LIN {X 0,Y 680.2,Z 809.06,A -85,B 0,C 180,E1 4290.744,E2 4290.744} C_VEL
LIN {X 0,Y 680.187,Z 809.06,A -85,B 0,C 180,E1 4295.606,E2 4295.606} C_VEL
LIN {X 0,Y 680.262,Z 809.06,A -85,B 0,C 180,E1 4300.538,E2 4300.538} C_VEL
LIN {X 0,Y 680.314,Z 809.425,A -85,B 0,C 180,E1 4305.507,E2 4305.507} C_VEL
LIN {X 0,Y 694.764,Z 845.315,A -85,B 0,C 180,E1 4307.71,E2 4307.71} C_VEL
LIN {X 0,Y 692.334,Z 893.553,A -85,B 0,C 180,E1 4309.75,E2 4309.75} C_VEL
LIN {X 0,Y 689.663,Z 937.812,A -85,B 0,C 180,E1 4312.208,E2 4312.208} C_VEL
LIN {X 0,Y 687.125,Z 980.915,A -85,B 0,C 180,E1 4315.269,E2 4315.269} C_VEL
LIN {X 0,Y 684.876,Z 1019.676,A -85,B 0,C 180,E1 4318.735,E2 4318.735} C_VEL
LIN {X 0,Y 683.218,Z 1052.318,A -85,B 0,C 180,E1 4322.376,E2 4322.376} C_VEL
LIN {X 0,Y 682.033,Z 1079.766,A -85,B 0,C 180,E1 4326.2,E2 4326.2} C_VEL
LIN {X 0,Y 681.334,Z 1102.128,A -85,B 0,C 180,E1 4330.219,E2 4330.219} C_VEL
LIN {X 0,Y 680.855,Z 1118.33,A -85,B 0,C 180,E1 4334.129,E2 4334.129} C_VEL
LIN {X 0,Y 680.765,Z 1129.59,A -85,B 0,C 180,E1 4338.103,E2 4338.103} C_VEL
LIN {X 0,Y 680.55,Z 1135.714,A -85,B 0,C 180,E1 4342.175,E2 4342.175} C_VEL
LIN {X 0,Y 680.543,Z 1137,A -85,B 0,C 180,E1 4344.951,E2 4344.951} C_VEL
LIN {X 0,Y 680.663,Z 1134.112,A -85,B 0,C 180,E1 4349.233,E2 4349.233} C_VEL
LIN {X 0,Y 680.799,Z 1126.558,A -85,B 0,C 180,E1 4353.076,E2 4353.076} C_VEL
LIN {X 0,Y 680.997,Z 1113.936,A -85,B 0,C 180,E1 4356.994,E2 4356.994} C_VEL
LIN {X 0,Y 681.399,Z 1096.802,A -85,B 0,C 180,E1 4360.757,E2 4360.757} C_VEL
LIN {X 0,Y 682.358,Z 1072.024,A -85,B 0,C 180,E1 4364.884,E2 4364.884} C_VEL
LIN {X 0,Y 683.721,Z 1042.519,A -85,B 0,C 180,E1 4368.71,E2 4368.71} C_VEL
LIN {X 0,Y 685.454,Z 1008.675,A -85,B 0,C 180,E1 4372.241,E2 4372.241} C_VEL
LIN {X 0,Y 687.791,Z 969.225,A -85,B 0,C 180,E1 4375.541,E2 4375.541} C_VEL
LIN {X 0,Y 690.35,Z 927.638,A -85,B 0,C 180,E1 4378.317,E2 4378.317} C_VEL
LIN {X 0,Y 692.87,Z 881.741,A -85,B 0,C 180,E1 4380.727,E2 4380.727} C_VEL
LIN {X 0,Y 694.585,Z 843.173,A -85,B 0,C 180,E1 4382.295,E2 4382.295} C_VEL
LIN {X 0,Y 680.289,Z 809.06,A -85,B 0,C 180,E1 4384.475,E2 4384.475} C_VEL
LIN {X 0,Y 680.236,Z 809.06,A -85,B 0,C 180,E1 4389.187,E2 4389.187} C_VEL
LIN {X 0,Y 680.252,Z 809.06,A -85,B 0,C 180,E1 4394.546,E2 4394.546} C_VEL
LIN {X 0,Y 680.62,Z 809.06,A -85,B 0,C 180,E1 4399.775,E2 4399.775} C_VEL
LIN {X 0,Y 680.649,Z 809.06,A -85,B 0,C 180,E1 4404.911,E2 4404.911} C_VEL
LIN {X 0,Y 680.652,Z 809.06,A -85,B 0,C 180,E1 4410.005,E2 4410.005} C_VEL
LIN {X 0,Y 680.742,Z 809.06,A -85,B 0,C 180,E1 4415.099,E2 4415.099} C_VEL
LIN {X 0,Y 680.549,Z 809.06,A -85,B 0,C 180,E1 4420.237,E2 4420.237} C_VEL
LIN {X 0,Y 680.532,Z 809.06,A -85,B 0,C 180,E1 4425.458,E2 4425.458} C_VEL
LIN {X 0,Y 680.453,Z 809.06,A -85,B 0,C 180,E1 4430.818,E2 4430.818} C_VEL
LIN {X 0,Y 680.319,Z 809.06,A -85,B 0,C 180,E1 4436.379,E2 4436.379} C_VEL
LIN {X 0,Y 680.313,Z 809.06,A -85,B 0,C 180,E1 4440.727,E2 4440.727} C_VEL
LIN {X 0,Y 680.298,Z 809.06,A -85,B 0,C 180,E1 4445.281,E2 4445.281} C_VEL
LIN {X 0,Y 680.16,Z 809.06,A -85,B 0,C 180,E1 4450.948,E2 4450.948} C_VEL
LIN {X 0,Y 680.352,Z 809.06,A -85,B 0,C 180,E1 4455.3,E2 4455.3} C_VEL
LIN {X 0,Y 680.213,Z 809.06,A -85,B 0,C 180,E1 4461.04,E2 4461.04} C_VEL
LIN {X 0,Y 680.177,Z 809.06,A -85,B 0,C 180,E1 4466.265,E2 4466.265} C_VEL
LIN {X 0,Y 680.337,Z 809.06,A -85,B 0,C 180,E1 4470.751,E2 4470.751} C_VEL
LIN {X 0,Y 680.434,Z 809.06,A -85,B 0,C 180,E1 4475.586,E2 4475.586} C_VEL
LIN {X 0,Y 680.513,Z 809.06,A -85,B 0,C 180,E1 4480.546,E2 4480.546} C_VEL
LIN {X 0,Y 680.474,Z 809.06,A -85,B 0,C 180,E1 4485.863,E2 4485.863} C_VEL
LIN {X 0,Y 680.596,Z 809.06,A -85,B 0,C 180,E1 4491.06,E2 4491.06} C_VEL
LIN {X 0,Y 680.727,Z 809.06,A -85,B 0,C 180,E1 4496.182,E2 4496.182} C_VEL
LIN {X 0,Y 680.902,Z 809.06,A -85,B 0,C 180,E1 4501.272,E2 4501.272} C_VEL
LIN {X 0,Y 680.599,Z 809.06,A -85,B 0,C 180,E1 4506.374,E2 4506.374} C_VEL
LIN {X 0,Y 680.537,Z 809.06,A -85,B 0,C 180,E1 4511.527,E2 4511.527} C_VEL
LIN {X 0,Y 680.557,Z 809.06,A -85,B 0,C 180,E1 4516.776,E2 4516.776} C_VEL
LIN {X 0,Y 680.391,Z 809.06,A -85,B 0,C 180,E1 4522.181,E2 4522.181} C_VEL
LIN {X 0,Y 680.331,Z 809.06,A -85,B 0,C 180,E1 4522.927,E2 4522.927} C_VEL
LIN {X 0,Y 676.369,Z 809.06,A -85,B 0,C 180,E1 4524.36,E2 4524.36} C_VEL
LIN {X 0,Y 672.401,Z 809.06,A -85,B 0,C 180,E1 4525.811,E2 4525.811} C_VEL
LIN {X 0,Y 672.352,Z 809.06,A -85,B 0,C 180,E1 4531.339,E2 4531.339} C_VEL
LIN {X 0,Y 672.336,Z 809.06,A -85,B 0,C 180,E1 4535.985,E2 4535.985} C_VEL
LIN {X 0,Y 672.291,Z 809.06,A -85,B 0,C 180,E1 4540.677,E2 4540.677} C_VEL
LIN {X 0,Y 672.415,Z 809.06,A -85,B 0,C 180,E1 4545.979,E2 4545.979} C_VEL
LIN {X 0,Y 672.345,Z 809.06,A -85,B 0,C 180,E1 4547.281,E2 4547.281} C_VEL
LIN {X 0,Y 674.931,Z 814.91,A -85,B 0,C 180,E1 4547.589,E2 4547.589} C_VEL
LIN {X 0,Y 692.454,Z 845.695,A -85,B 0,C 180,E1 4549.313,E2 4549.313} C_VEL
LIN {X 0,Y 691.569,Z 922.86,A -85,B 0,C 180,E1 4550.398,E2 4550.398} C_VEL
LIN {X 0,Y 689.719,Z 966.962,A -85,B 0,C 180,E1 4551.427,E2 4551.427} C_VEL
LIN {X 0,Y 687.547,Z 1012.993,A -85,B 0,C 180,E1 4553.033,E2 4553.033} C_VEL
LIN {X 0,Y 684.845,Z 1057.118,A -85,B 0,C 180,E1 4555.103,E2 4555.103} C_VEL
LIN {X 0,Y 682.1,Z 1099.687,A -85,B 0,C 180,E1 4557.663,E2 4557.663} C_VEL
LIN {X 0,Y 679.28,Z 1140.676,A -85,B 0,C 180,E1 4560.788,E2 4560.788} C_VEL
LIN {X 0,Y 677.093,Z 1175.037,A -85,B 0,C 180,E1 4564.02,E2 4564.02} C_VEL
LIN {X 0,Y 675.283,Z 1208.242,A -85,B 0,C 180,E1 4567.912,E2 4567.912} C_VEL
LIN {X 0,Y 674.008,Z 1233.927,A -85,B 0,C 180,E1 4571.702,E2 4571.702} C_VEL
LIN {X 0,Y 673.404,Z 1254.994,A -85,B 0,C 180,E1 4575.705,E2 4575.705} C_VEL
LIN {X 0,Y 673.092,Z 1270.402,A -85,B 0,C 180,E1 4579.649,E2 4579.649} C_VEL
LIN {X 0,Y 672.976,Z 1280.56,A -85,B 0,C 180,E1 4583.549,E2 4583.549} C_VEL
LIN {X 0,Y 672.892,Z 1285.871,A -85,B 0,C 180,E1 4587.421,E2 4587.421} C_VEL
LIN {X 0,Y 673.007,Z 1286.67,A -85,B 0,C 180,E1 4591.281,E2 4591.281} C_VEL
LIN {X 0,Y 672.834,Z 1282.919,A -85,B 0,C 180,E1 4595.149,E2 4595.149} C_VEL
LIN {X 0,Y 672.864,Z 1274.306,A -85,B 0,C 180,E1 4599.039,E2 4599.039} C_VEL
LIN {X 0,Y 673.22,Z 1262.369,A -85,B 0,C 180,E1 4602.563,E2 4602.563} C_VEL
LIN {X 0,Y 673.685,Z 1243.504,A -85,B 0,C 180,E1 4606.612,E2 4606.612} C_VEL
LIN {X 0,Y 674.721,Z 1219.785,A -85,B 0,C 180,E1 4610.494,E2 4610.494} C_VEL
LIN {X 0,Y 676.337,Z 1189.33,A -85,B 0,C 180,E1 4614.408,E2 4614.408} C_VEL
LIN {X 0,Y 678.339,Z 1155.606,A -85,B 0,C 180,E1 4617.885,E2 4617.885} C_VEL
LIN {X 0,Y 680.944,Z 1116.496,A -85,B 0,C 180,E1 4621.144,E2 4621.144} C_VEL
LIN {X 0,Y 683.675,Z 1073.955,A -85,B 0,C 180,E1 4623.959,E2 4623.959} C_VEL
LIN {X 0,Y 686.596,Z 1029.232,A -85,B 0,C 180,E1 4626.275,E2 4626.275} C_VEL
LIN {X 0,Y 689.056,Z 982.863,A -85,B 0,C 180,E1 4628.07,E2 4628.07} C_VEL
LIN {X 0,Y 691.01,Z 936.03,A -85,B 0,C 180,E1 4629.35,E2 4629.35} C_VEL
LIN {X 0,Y 692.232,Z 887.052,A -85,B 0,C 180,E1 4630.15,E2 4630.15} C_VEL
LIN {X 0,Y 691.991,Z 845.459,A -85,B 0,C 180,E1 4630.723,E2 4630.723} C_VEL
LIN {X 0,Y 672.601,Z 810.385,A -85,B 0,C 180,E1 4632.657,E2 4632.657} C_VEL
LIN {X 0,Y 672.495,Z 809.06,A -85,B 0,C 180,E1 4632.782,E2 4632.782} C_VEL
LIN {X 0,Y 672.304,Z 809.06,A -85,B 0,C 180,E1 4637.868,E2 4637.868} C_VEL
LIN {X 0,Y 672.275,Z 809.06,A -85,B 0,C 180,E1 4642.638,E2 4642.638} C_VEL
LIN {X 0,Y 672.238,Z 809.06,A -85,B 0,C 180,E1 4647.353,E2 4647.353} C_VEL
LIN {X 0,Y 672.328,Z 809.06,A -85,B 0,C 180,E1 4651.838,E2 4651.838} C_VEL
LIN {X 0,Y 672.2,Z 809.06,A -85,B 0,C 180,E1 4657.154,E2 4657.154} C_VEL
LIN {X 0,Y 672.233,Z 809.06,A -85,B 0,C 180,E1 4661.658,E2 4661.658} C_VEL
LIN {X 0,Y 672.415,Z 809.64,A -85,B 0,C 180,E1 4664.957,E2 4664.957} C_VEL
LIN {X 0,Y 688.239,Z 847.852,A -85,B 0,C 180,E1 4667.398,E2 4667.398} C_VEL
LIN {X 0,Y 685.564,Z 895.468,A -85,B 0,C 180,E1 4669.452,E2 4669.452} C_VEL
LIN {X 0,Y 682.602,Z 939.865,A -85,B 0,C 180,E1 4671.967,E2 4671.967} C_VEL
LIN {X 0,Y 679.837,Z 982.551,A -85,B 0,C 180,E1 4675.059,E2 4675.059} C_VEL
LIN {X 0,Y 677.362,Z 1021.021,A -85,B 0,C 180,E1 4678.562,E2 4678.562} C_VEL
LIN {X 0,Y 675.566,Z 1053.378,A -85,B 0,C 180,E1 4682.243,E2 4682.243} C_VEL
LIN {X 0,Y 674.272,Z 1080.621,A -85,B 0,C 180,E1 4686.11,E2 4686.11} C_VEL
LIN {X 0,Y 673.504,Z 1102.103,A -85,B 0,C 180,E1 4690.038,E2 4690.038} C_VEL
LIN {X 0,Y 673.032,Z 1118.204,A -85,B 0,C 180,E1 4693.965,E2 4693.965} C_VEL
LIN {X 0,Y 672.892,Z 1128.636,A -85,B 0,C 180,E1 4697.604,E2 4697.604} C_VEL
LIN {X 0,Y 672.719,Z 1134.648,A -85,B 0,C 180,E1 4701.061,E2 4701.061} C_VEL
LIN {X 0,Y 672.605,Z 1136.938,A -85,B 0,C 180,E1 4705.266,E2 4705.266} C_VEL
LIN {X 0,Y 672.791,Z 1133.635,A -85,B 0,C 180,E1 4709.609,E2 4709.609} C_VEL
LIN {X 0,Y 672.957,Z 1126.007,A -85,B 0,C 180,E1 4713.387,E2 4713.387} C_VEL
LIN {X 0,Y 673.212,Z 1113.275,A -85,B 0,C 180,E1 4717.3,E2 4717.3} C_VEL
LIN {X 0,Y 673.741,Z 1094.48,A -85,B 0,C 180,E1 4721.384,E2 4721.384} C_VEL
LIN {X 0,Y 674.716,Z 1070.906,A -85,B 0,C 180,E1 4725.291,E2 4725.291} C_VEL
LIN {X 0,Y 676.283,Z 1041.021,A -85,B 0,C 180,E1 4729.166,E2 4729.166} C_VEL
LIN {X 0,Y 678.193,Z 1007.742,A -85,B 0,C 180,E1 4732.647,E2 4732.647} C_VEL
LIN {X 0,Y 680.795,Z 968.271,A -85,B 0,C 180,E1 4735.965,E2 4735.965} C_VEL
LIN {X 0,Y 683.603,Z 926.623,A -85,B 0,C 180,E1 4738.754,E2 4738.754} C_VEL
LIN {X 0,Y 686.379,Z 880.658,A -85,B 0,C 180,E1 4741.173,E2 4741.173} C_VEL
LIN {X 0,Y 687.87,Z 845.761,A -85,B 0,C 180,E1 4742.623,E2 4742.623} C_VEL
LIN {X 0,Y 672.359,Z 809.06,A -85,B 0,C 180,E1 4745.019,E2 4745.019} C_VEL
LIN {X 0,Y 672.331,Z 809.06,A -85,B 0,C 180,E1 4750.716,E2 4750.716} C_VEL
LIN {X 0,Y 672.433,Z 809.06,A -85,B 0,C 180,E1 4755.694,E2 4755.694} C_VEL
LIN {X 0,Y 672.681,Z 809.06,A -85,B 0,C 180,E1 4760.959,E2 4760.959} C_VEL
LIN {X 0,Y 672.768,Z 809.06,A -85,B 0,C 180,E1 4766.142,E2 4766.142} C_VEL
LIN {X 0,Y 672.896,Z 809.06,A -85,B 0,C 180,E1 4771.292,E2 4771.292} C_VEL
LIN {X 0,Y 672.654,Z 809.06,A -85,B 0,C 180,E1 4776.454,E2 4776.454} C_VEL
LIN {X 0,Y 672.629,Z 809.06,A -85,B 0,C 180,E1 4781.67,E2 4781.67} C_VEL
LIN {X 0,Y 672.673,Z 809.06,A -85,B 0,C 180,E1 4786.985,E2 4786.985} C_VEL
LIN {X 0,Y 672.468,Z 809.06,A -85,B 0,C 180,E1 4792.463,E2 4792.463} C_VEL
LIN {X 0,Y 672.432,Z 809.06,A -85,B 0,C 180,E1 4796.713,E2 4796.713} C_VEL
LIN {X 0,Y 672.367,Z 809.06,A -85,B 0,C 180,E1 4801.356,E2 4801.356} C_VEL
LIN {X 0,Y 672.334,Z 809.06,A -85,B 0,C 180,E1 4805.997,E2 4805.997} C_VEL
LIN {X 0,Y 672.257,Z 809.06,A -85,B 0,C 180,E1 4810.687,E2 4810.687} C_VEL
LIN {X 0,Y 672.372,Z 809.06,A -85,B 0,C 180,E1 4815.842,E2 4815.842} C_VEL
LIN {X 0,Y 672.317,Z 809.06,A -85,B 0,C 180,E1 4821.003,E2 4821.003} C_VEL
LIN {X 0,Y 672.287,Z 809.06,A -85,B 0,C 180,E1 4826.275,E2 4826.275} C_VEL
LIN {X 0,Y 672.481,Z 809.06,A -85,B 0,C 180,E1 4831.846,E2 4831.846} C_VEL
LIN {X 0,Y 672.489,Z 809.06,A -85,B 0,C 180,E1 4837.122,E2 4837.122} C_VEL
LIN {X 0,Y 672.603,Z 809.06,A -85,B 0,C 180,E1 4841.669,E2 4841.669} C_VEL
LIN {X 0,Y 672.519,Z 809.06,A -85,B 0,C 180,E1 4847.017,E2 4847.017} C_VEL
LIN {X 0,Y 672.766,Z 809.06,A -85,B 0,C 180,E1 4852.256,E2 4852.256} C_VEL
LIN {X 0,Y 672.902,Z 809.06,A -85,B 0,C 180,E1 4857.426,E2 4857.426} C_VEL
LIN {X 0,Y 672.764,Z 809.06,A -85,B 0,C 180,E1 4862.575,E2 4862.575} C_VEL
LIN {X 0,Y 672.691,Z 809.06,A -85,B 0,C 180,E1 4866.449,E2 4866.449} C_VEL
LIN {X 0,Y 672.682,Z 809.06,A -85,B 0,C 180,E1 4870.353,E2 4870.353} C_VEL
LIN {X 0,Y 672.606,Z 809.06,A -85,B 0,C 180,E1 4875.64,E2 4875.64} C_VEL
LIN {X 0,Y 672.538,Z 809.06,A -85,B 0,C 180,E1 4881.068,E2 4881.068} C_VEL
LIN {X 0,Y 672.401,Z 809.06,A -85,B 0,C 180,E1 4885.811,E2 4885.811} C_VEL
LIN {X 0,Y 668.475,Z 809.06,A -85,B 0,C 180,E1 4887.268,E2 4887.268} C_VEL
LIN {X 0,Y 664.434,Z 809.06,A -85,B 0,C 180,E1 4888.742,E2 4888.742} C_VEL
LIN {X 0,Y 664.486,Z 809.06,A -85,B 0,C 180,E1 4893.076,E2 4893.076} C_VEL
LIN {X 0,Y 664.378,Z 809.06,A -85,B 0,C 180,E1 4897.884,E2 4897.884} C_VEL
LIN {X 0,Y 664.506,Z 809.06,A -85,B 0,C 180,E1 4903.302,E2 4903.302} C_VEL
LIN {X 0,Y 664.45,Z 809.06,A -85,B 0,C 180,E1 4906.65,E2 4906.65} C_VEL
LIN {X 0,Y 666.896,Z 814.808,A -85,B 0,C 180,E1 4906.953,E2 4906.953} C_VEL
LIN {X 0,Y 686.477,Z 848.997,A -85,B 0,C 180,E1 4908.928,E2 4908.928} C_VEL
LIN {X 0,Y 685.465,Z 922.835,A -85,B 0,C 180,E1 4909.974,E2 4909.974} C_VEL
LIN {X 0,Y 683.47,Z 967.502,A -85,B 0,C 180,E1 4911.026,E2 4911.026} C_VEL
LIN {X 0,Y 681.085,Z 1013.115,A -85,B 0,C 180,E1 4912.629,E2 4912.629} C_VEL
LIN {X 0,Y 678.207,Z 1056.587,A -85,B 0,C 180,E1 4914.68,E2 4914.68} C_VEL
LIN {X 0,Y 675.251,Z 1098.141,A -85,B 0,C 180,E1 4917.187,E2 4917.187} C_VEL
LIN {X 0,Y 672.226,Z 1138.223,A -85,B 0,C 180,E1 4920.234,E2 4920.234} C_VEL
LIN {X 0,Y 669.782,Z 1173.415,A -85,B 0,C 180,E1 4923.535,E2 4923.535} C_VEL
LIN {X 0,Y 667.651,Z 1206.126,A -85,B 0,C 180,E1 4927.366,E2 4927.366} C_VEL
LIN {X 0,Y 666.283,Z 1231.954,A -85,B 0,C 180,E1 4931.14,E2 4931.14} C_VEL
LIN {X 0,Y 665.611,Z 1251.057,A -85,B 0,C 180,E1 4934.679,E2 4934.679} C_VEL
LIN {X 0,Y 665.138,Z 1266.966,A -85,B 0,C 180,E1 4938.529,E2 4938.529} C_VEL
LIN {X 0,Y 664.972,Z 1277.702,A -85,B 0,C 180,E1 4942.158,E2 4942.158} C_VEL
LIN {X 0,Y 664.985,Z 1284.672,A -85,B 0,C 180,E1 4946.086,E2 4946.086} C_VEL
LIN {X 0,Y 664.95,Z 1287,A -85,B 0,C 180,E1 4949.995,E2 4949.995} C_VEL
LIN {X 0,Y 665.027,Z 1284.685,A -85,B 0,C 180,E1 4953.903,E2 4953.903} C_VEL
LIN {X 0,Y 664.965,Z 1277.728,A -85,B 0,C 180,E1 4957.831,E2 4957.831} C_VEL
LIN {X 0,Y 665.261,Z 1265.849,A -85,B 0,C 180,E1 4961.79,E2 4961.79} C_VEL
LIN {X 0,Y 665.675,Z 1248.748,A -85,B 0,C 180,E1 4965.801,E2 4965.801} C_VEL
LIN {X 0,Y 666.57,Z 1227.725,A -85,B 0,C 180,E1 4969.528,E2 4969.528} C_VEL
LIN {X 0,Y 668.057,Z 1199.843,A -85,B 0,C 180,E1 4973.444,E2 4973.444} C_VEL
LIN {X 0,Y 670.119,Z 1168.064,A -85,B 0,C 180,E1 4977.004,E2 4977.004} C_VEL
LIN {X 0,Y 672.789,Z 1131.27,A -85,B 0,C 180,E1 4980.354,E2 4980.354} C_VEL
LIN {X 0,Y 675.867,Z 1089.063,A -85,B 0,C 180,E1 4983.409,E2 4983.409} C_VEL
LIN {X 0,Y 678.951,Z 1046.719,A -85,B 0,C 180,E1 4985.837,E2 4985.837} C_VEL
LIN {X 0,Y 681.717,Z 1002.725,A -85,B 0,C 180,E1 4987.775,E2 4987.775} C_VEL
LIN {X 0,Y 684.002,Z 957.416,A -85,B 0,C 180,E1 4989.252,E2 4989.252} C_VEL
LIN {X 0,Y 685.728,Z 911.796,A -85,B 0,C 180,E1 4990.23,E2 4990.23} C_VEL
LIN {X 0,Y 686.126,Z 848.928,A -85,B 0,C 180,E1 4991.099,E2 4991.099} C_VEL
LIN {X 0,Y 664.669,Z 810.286,A -85,B 0,C 180,E1 4993.292,E2 4993.292} C_VEL
LIN {X 0,Y 664.559,Z 809.06,A -85,B 0,C 180,E1 4993.448,E2 4993.448} C_VEL
LIN {X 0,Y 664.342,Z 809.06,A -85,B 0,C 180,E1 4998.731,E2 4998.731} C_VEL
LIN {X 0,Y 664.376,Z 809.06,A -85,B 0,C 180,E1 5003.749,E2 5003.749} C_VEL
LIN {X 0,Y 664.333,Z 809.06,A -85,B 0,C 180,E1 5008.458,E2 5008.458} C_VEL
LIN {X 0,Y 664.421,Z 809.06,A -85,B 0,C 180,E1 5012.946,E2 5012.946} C_VEL
LIN {X 0,Y 664.412,Z 809.06,A -85,B 0,C 180,E1 5018.804,E2 5018.804} C_VEL
LIN {X 0,Y 664.425,Z 809.363,A -85,B 0,C 180,E1 5024.368,E2 5024.368} C_VEL
LIN {X 0,Y 681.715,Z 851.229,A -85,B 0,C 180,E1 5027.114,E2 5027.114} C_VEL
LIN {X 0,Y 678.769,Z 897.923,A -85,B 0,C 180,E1 5029.174,E2 5029.174} C_VEL
LIN {X 0,Y 675.505,Z 943.111,A -85,B 0,C 180,E1 5031.801,E2 5031.801} C_VEL
LIN {X 0,Y 672.55,Z 984.171,A -85,B 0,C 180,E1 5034.844,E2 5034.844} C_VEL
LIN {X 0,Y 669.858,Z 1022.355,A -85,B 0,C 180,E1 5038.384,E2 5038.384} C_VEL
LIN {X 0,Y 667.884,Z 1054.448,A -85,B 0,C 180,E1 5042.106,E2 5042.106} C_VEL
LIN {X 0,Y 666.543,Z 1080.442,A -85,B 0,C 180,E1 5045.854,E2 5045.854} C_VEL
LIN {X 0,Y 665.705,Z 1101.84,A -85,B 0,C 180,E1 5049.801,E2 5049.801} C_VEL
LIN {X 0,Y 665.167,Z 1118.084,A -85,B 0,C 180,E1 5053.799,E2 5053.799} C_VEL
LIN {X 0,Y 664.972,Z 1129.577,A -85,B 0,C 180,E1 5057.934,E2 5057.934} C_VEL
LIN {X 0,Y 664.799,Z 1135.004,A -85,B 0,C 180,E1 5061.324,E2 5061.324} C_VEL
LIN {X 0,Y 664.704,Z 1136.864,A -85,B 0,C 180,E1 5065.588,E2 5065.588} C_VEL
LIN {X 0,Y 664.776,Z 1135.08,A -85,B 0,C 180,E1 5068.51,E2 5068.51} C_VEL
LIN {X 0,Y 665.011,Z 1128.8,A -85,B 0,C 180,E1 5072.323,E2 5072.323} C_VEL
LIN {X 0,Y 665.166,Z 1117.778,A -85,B 0,C 180,E1 5076.2,E2 5076.2} C_VEL
LIN {X 0,Y 665.561,Z 1103.198,A -85,B 0,C 180,E1 5079.816,E2 5079.816} C_VEL
LIN {X 0,Y 666.338,Z 1082.447,A -85,B 0,C 180,E1 5083.726,E2 5083.726} C_VEL
LIN {X 0,Y 667.692,Z 1056.685,A -85,B 0,C 180,E1 5087.519,E2 5087.519} C_VEL
LIN {X 0,Y 669.71,Z 1024.273,A -85,B 0,C 180,E1 5091.327,E2 5091.327} C_VEL
LIN {X 0,Y 672.295,Z 987.168,A -85,B 0,C 180,E1 5094.817,E2 5094.817} C_VEL
LIN {X 0,Y 675.29,Z 947.344,A -85,B 0,C 180,E1 5097.821,E2 5097.821} C_VEL
LIN {X 0,Y 678.42,Z 904.103,A -85,B 0,C 180,E1 5100.411,E2 5100.411} C_VEL
LIN {X 0,Y 681.233,Z 861.151,A -85,B 0,C 180,E1 5102.405,E2 5102.405} C_VEL
LIN {X 0,Y 681.663,Z 849.788,A -85,B 0,C 180,E1 5102.861,E2 5102.861} C_VEL
LIN {X 0,Y 664.402,Z 809.06,A -85,B 0,C 180,E1 5105.602,E2 5105.602} C_VEL
LIN {X 0,Y 664.404,Z 809.06,A -85,B 0,C 180,E1 5110.059,E2 5110.059} C_VEL
LIN {X 0,Y 664.518,Z 809.06,A -85,B 0,C 180,E1 5115.52,E2 5115.52} C_VEL
LIN {X 0,Y 664.771,Z 809.06,A -85,B 0,C 180,E1 5120.85,E2 5120.85} C_VEL
LIN {X 0,Y 664.88,Z 809.06,A -85,B 0,C 180,E1 5126.096,E2 5126.096} C_VEL
LIN {X 0,Y 665.002,Z 809.06,A -85,B 0,C 180,E1 5131.307,E2 5131.307} C_VEL
LIN {X 0,Y 664.755,Z 809.06,A -85,B 0,C 180,E1 5136.531,E2 5136.531} C_VEL
LIN {X 0,Y 664.716,Z 809.06,A -85,B 0,C 180,E1 5141.811,E2 5141.811} C_VEL
LIN {X 0,Y 664.725,Z 809.06,A -85,B 0,C 180,E1 5147.313,E2 5147.313} C_VEL
LIN {X 0,Y 664.556,Z 809.06,A -85,B 0,C 180,E1 5152.745,E2 5152.745} C_VEL
LIN {X 0,Y 664.504,Z 809.06,A -85,B 0,C 180,E1 5157.527,E2 5157.527} C_VEL
LIN {X 0,Y 664.521,Z 809.06,A -85,B 0,C 180,E1 5163.081,E2 5163.081} C_VEL
LIN {X 0,Y 664.36,Z 809.06,A -85,B 0,C 180,E1 5167.893,E2 5167.893} C_VEL
LIN {X 0,Y 664.475,Z 809.06,A -85,B 0,C 180,E1 5173.31,E2 5173.31} C_VEL
LIN {X 0,Y 664.317,Z 809.06,A -85,B 0,C 180,E1 5178.731,E2 5178.731} C_VEL
LIN {X 0,Y 664.359,Z 809.06,A -85,B 0,C 180,E1 5183.749,E2 5183.749} C_VEL
LIN {X 0,Y 664.381,Z 809.06,A -85,B 0,C 180,E1 5188.461,E2 5188.461} C_VEL
LIN {X 0,Y 664.609,Z 809.06,A -85,B 0,C 180,E1 5192.955,E2 5192.955} C_VEL
LIN {X 0,Y 664.634,Z 809.06,A -85,B 0,C 180,E1 5198.67,E2 5198.67} C_VEL
LIN {X 0,Y 664.686,Z 809.06,A -85,B 0,C 180,E1 5204.17,E2 5204.17} C_VEL
LIN {X 0,Y 664.804,Z 809.06,A -85,B 0,C 180,E1 5209.524,E2 5209.524} C_VEL
LIN {X 0,Y 664.815,Z 809.06,A -85,B 0,C 180,E1 5214.784,E2 5214.784} C_VEL
LIN {X 0,Y 664.929,Z 809.06,A -85,B 0,C 180,E1 5219.708,E2 5219.708} C_VEL
LIN {X 0,Y 664.955,Z 809.06,A -85,B 0,C 180,E1 5223.909,E2 5223.909} C_VEL
LIN {X 0,Y 664.854,Z 809.06,A -85,B 0,C 180,E1 5229.154,E2 5229.154} C_VEL
LIN {X 0,Y 664.687,Z 809.06,A -85,B 0,C 180,E1 5234.481,E2 5234.481} C_VEL
LIN {X 0,Y 664.679,Z 809.06,A -85,B 0,C 180,E1 5238.558,E2 5238.558} C_VEL
LIN {X 0,Y 664.548,Z 809.06,A -85,B 0,C 180,E1 5242.739,E2 5242.739} C_VEL
LIN {X 0,Y 664.443,Z 809.06,A -85,B 0,C 180,E1 5247.5,E2 5247.5} C_VEL
LIN {X 0,Y 664.434,Z 809.06,A -85,B 0,C 180,E1 5248.742,E2 5248.742} C_VEL
LIN {X 0,Y 660.457,Z 809.06,A -85,B 0,C 180,E1 5250.217,E2 5250.217} C_VEL
LIN {X 0,Y 656.542,Z 809.06,A -85,B 0,C 180,E1 5251.709,E2 5251.709} C_VEL
LIN {X 0,Y 656.493,Z 809.06,A -85,B 0,C 180,E1 5256.757,E2 5256.757} C_VEL
LIN {X 0,Y 656.531,Z 809.06,A -85,B 0,C 180,E1 5262.558,E2 5262.558} C_VEL
LIN {X 0,Y 656.603,Z 809.06,A -85,B 0,C 180,E1 5266.019,E2 5266.019} C_VEL
LIN {X 0,Y 659.009,Z 814.762,A -85,B 0,C 180,E1 5266.309,E2 5266.309} C_VEL
LIN {X 0,Y 680.523,Z 852.366,A -85,B 0,C 180,E1 5268.536,E2 5268.536} C_VEL
LIN {X 0,Y 679.352,Z 923.994,A -85,B 0,C 180,E1 5269.565,E2 5269.565} C_VEL
LIN {X 0,Y 677.255,Z 967.989,A -85,B 0,C 180,E1 5270.615,E2 5270.615} C_VEL
LIN {X 0,Y 674.723,Z 1012.719,A -85,B 0,C 180,E1 5272.196,E2 5272.196} C_VEL
LIN {X 0,Y 671.609,Z 1056.2,A -85,B 0,C 180,E1 5274.258,E2 5274.258} C_VEL
LIN {X 0,Y 668.269,Z 1098.966,A -85,B 0,C 180,E1 5276.858,E2 5276.858} C_VEL
LIN {X 0,Y 664.943,Z 1139.603,A -85,B 0,C 180,E1 5279.998,E2 5279.998} C_VEL
LIN {X 0,Y 662.248,Z 1175.04,A -85,B 0,C 180,E1 5283.393,E2 5283.393} C_VEL
LIN {X 0,Y 659.946,Z 1207.625,A -85,B 0,C 180,E1 5287.289,E2 5287.289} C_VEL
LIN {X 0,Y 658.545,Z 1232.261,A -85,B 0,C 180,E1 5290.963,E2 5290.963} C_VEL
LIN {X 0,Y 657.726,Z 1252.321,A -85,B 0,C 180,E1 5294.768,E2 5294.768} C_VEL
LIN {X 0,Y 657.282,Z 1268.123,A -85,B 0,C 180,E1 5298.726,E2 5298.726} C_VEL
LIN {X 0,Y 657.129,Z 1279.211,A -85,B 0,C 180,E1 5302.729,E2 5302.729} C_VEL
LIN {X 0,Y 657.08,Z 1284.672,A -85,B 0,C 180,E1 5306.039,E2 5306.039} C_VEL
LIN {X 0,Y 657.075,Z 1287,A -85,B 0,C 180,E1 5309.995,E2 5309.995} C_VEL
LIN {X 0,Y 657.119,Z 1284.685,A -85,B 0,C 180,E1 5313.95,E2 5313.95} C_VEL
LIN {X 0,Y 657.07,Z 1277.725,A -85,B 0,C 180,E1 5317.926,E2 5317.926} C_VEL
LIN {X 0,Y 657.398,Z 1265.85,A -85,B 0,C 180,E1 5321.933,E2 5321.933} C_VEL
LIN {X 0,Y 657.839,Z 1249.826,A -85,B 0,C 180,E1 5325.778,E2 5325.778} C_VEL
LIN {X 0,Y 658.799,Z 1228.696,A -85,B 0,C 180,E1 5329.611,E2 5329.611} C_VEL
LIN {X 0,Y 660.348,Z 1201.517,A -85,B 0,C 180,E1 5333.512,E2 5333.512} C_VEL
LIN {X 0,Y 662.594,Z 1170.029,A -85,B 0,C 180,E1 5337.13,E2 5337.13} C_VEL
LIN {X 0,Y 665.676,Z 1131.248,A -85,B 0,C 180,E1 5340.715,E2 5340.715} C_VEL
LIN {X 0,Y 668.977,Z 1089.446,A -85,B 0,C 180,E1 5343.773,E2 5343.773} C_VEL
LIN {X 0,Y 672.36,Z 1046.704,A -85,B 0,C 180,E1 5346.245,E2 5346.245} C_VEL
LIN {X 0,Y 675.412,Z 1001.915,A -85,B 0,C 180,E1 5348.224,E2 5348.224} C_VEL
LIN {X 0,Y 677.847,Z 957.042,A -85,B 0,C 180,E1 5349.689,E2 5349.689} C_VEL
LIN {X 0,Y 679.724,Z 910.77,A -85,B 0,C 180,E1 5350.678,E2 5350.678} C_VEL
LIN {X 0,Y 680.189,Z 852.119,A -85,B 0,C 180,E1 5351.492,E2 5351.492} C_VEL
LIN {X 0,Y 656.877,Z 810.783,A -85,B 0,C 180,E1 5353.928,E2 5353.928} C_VEL
LIN {X 0,Y 656.682,Z 809.06,A -85,B 0,C 180,E1 5354.019,E2 5354.019} C_VEL
LIN {X 0,Y 656.404,Z 809.06,A -85,B 0,C 180,E1 5359.868,E2 5359.868} C_VEL
LIN {X 0,Y 656.433,Z 809.06,A -85,B 0,C 180,E1 5364.868,E2 5364.868} C_VEL
LIN {X 0,Y 656.424,Z 809.06,A -85,B 0,C 180,E1 5369.575,E2 5369.575} C_VEL
LIN {X 0,Y 656.491,Z 809.06,A -85,B 0,C 180,E1 5374.067,E2 5374.067} C_VEL
LIN {X 0,Y 656.516,Z 809.06,A -85,B 0,C 180,E1 5379.804,E2 5379.804} C_VEL
LIN {X 0,Y 656.454,Z 809.14,A -85,B 0,C 180,E1 5383.762,E2 5383.762} C_VEL
LIN {X 0,Y 675.009,Z 852.682,A -85,B 0,C 180,E1 5386.731,E2 5386.731} C_VEL
LIN {X 0,Y 671.989,Z 900.519,A -85,B 0,C 180,E1 5388.899,E2 5388.899} C_VEL
LIN {X 0,Y 668.407,Z 946.346,A -85,B 0,C 180,E1 5391.632,E2 5391.632} C_VEL
LIN {X 0,Y 665.282,Z 985.787,A -85,B 0,C 180,E1 5394.624,E2 5394.624} C_VEL
LIN {X 0,Y 662.477,Z 1022.118,A -85,B 0,C 180,E1 5398.039,E2 5398.039} C_VEL
LIN {X 0,Y 660.299,Z 1054.255,A -85,B 0,C 180,E1 5401.803,E2 5401.803} C_VEL
LIN {X 0,Y 658.776,Z 1081.294,A -85,B 0,C 180,E1 5405.759,E2 5405.759} C_VEL
LIN {X 0,Y 657.816,Z 1103.23,A -85,B 0,C 180,E1 5409.92,E2 5409.92} C_VEL
LIN {X 0,Y 657.269,Z 1119.137,A -85,B 0,C 180,E1 5413.968,E2 5413.968} C_VEL
LIN {X 0,Y 657.083,Z 1130.05,A -85,B 0,C 180,E1 5418.085,E2 5418.085} C_VEL
LIN {X 0,Y 656.848,Z 1135.326,A -85,B 0,C 180,E1 5421.595,E2 5421.595} C_VEL
LIN {X 0,Y 656.768,Z 1136.782,A -85,B 0,C 180,E1 5425.92,E2 5425.92} C_VEL
LIN {X 0,Y 657.077,Z 1132.658,A -85,B 0,C 180,E1 5430.391,E2 5430.391} C_VEL
LIN {X 0,Y 657.333,Z 1123.249,A -85,B 0,C 180,E1 5434.586,E2 5434.586} C_VEL
LIN {X 0,Y 657.69,Z 1107.865,A -85,B 0,C 180,E1 5438.948,E2 5438.948} C_VEL
LIN {X 0,Y 658.354,Z 1087.417,A -85,B 0,C 180,E1 5443.095,E2 5443.095} C_VEL
LIN {X 0,Y 659.813,Z 1061.64,A -85,B 0,C 180,E1 5447.122,E2 5447.122} C_VEL
LIN {X 0,Y 661.772,Z 1030.892,A -85,B 0,C 180,E1 5450.923,E2 5450.923} C_VEL
LIN {X 0,Y 664.441,Z 996.32,A -85,B 0,C 180,E1 5454.374,E2 5454.374} C_VEL
LIN {X 0,Y 667.578,Z 957.329,A -85,B 0,C 180,E1 5457.504,E2 5457.504} C_VEL
LIN {X 0,Y 670.863,Z 916.52,A -85,B 0,C 180,E1 5460.128,E2 5460.128} C_VEL
LIN {X 0,Y 673.925,Z 873.439,A -85,B 0,C 180,E1 5462.302,E2 5462.302} C_VEL
LIN {X 0,Y 674.788,Z 852.086,A -85,B 0,C 180,E1 5463.22,E2 5463.22} C_VEL
LIN {X 0,Y 658.078,Z 813.864,A -85,B 0,C 180,E1 5465.864,E2 5465.864} C_VEL
LIN {X 0,Y 656.419,Z 809.06,A -85,B 0,C 180,E1 5466.25,E2 5466.25} C_VEL
LIN {X 0,Y 656.429,Z 809.06,A -85,B 0,C 180,E1 5471.206,E2 5471.206} C_VEL
LIN {X 0,Y 656.655,Z 809.06,A -85,B 0,C 180,E1 5476.702,E2 5476.702} C_VEL
LIN {X 0,Y 656.916,Z 809.06,A -85,B 0,C 180,E1 5482.073,E2 5482.073} C_VEL
LIN {X 0,Y 657.028,Z 809.06,A -85,B 0,C 180,E1 5487.369,E2 5487.369} C_VEL
LIN {X 0,Y 656.898,Z 809.06,A -85,B 0,C 180,E1 5492.642,E2 5492.642} C_VEL
LIN {X 0,Y 656.849,Z 809.06,A -85,B 0,C 180,E1 5496.61,E2 5496.61} C_VEL
LIN {X 0,Y 656.827,Z 809.06,A -85,B 0,C 180,E1 5501.955,E2 5501.955} C_VEL
LIN {X 0,Y 656.827,Z 809.06,A -85,B 0,C 180,E1 5507.407,E2 5507.407} C_VEL
LIN {X 0,Y 656.644,Z 809.06,A -85,B 0,C 180,E1 5513.035,E2 5513.035} C_VEL
LIN {X 0,Y 656.597,Z 809.06,A -85,B 0,C 180,E1 5517.41,E2 5517.41} C_VEL
LIN {X 0,Y 656.553,Z 809.06,A -85,B 0,C 180,E1 5521.967,E2 5521.967} C_VEL
LIN {X 0,Y 656.48,Z 809.06,A -85,B 0,C 180,E1 5526.766,E2 5526.766} C_VEL
LIN {X 0,Y 656.498,Z 809.06,A -85,B 0,C 180,E1 5532.566,E2 5532.566} C_VEL
LIN {X 0,Y 656.393,Z 809.06,A -85,B 0,C 180,E1 5537.455,E2 5537.455} C_VEL
LIN {X 0,Y 656.423,Z 809.06,A -85,B 0,C 180,E1 5541.575,E2 5541.575} C_VEL
LIN {X 0,Y 656.394,Z 809.06,A -85,B 0,C 180,E1 5546.464,E2 5546.464} C_VEL
LIN {X 0,Y 656.569,Z 809.06,A -85,B 0,C 180,E1 5551.101,E2 5551.101} C_VEL
LIN {X 0,Y 656.695,Z 809.06,A -85,B 0,C 180,E1 5555.534,E2 5555.534} C_VEL
LIN {X 0,Y 656.759,Z 809.06,A -85,B 0,C 180,E1 5561.211,E2 5561.211} C_VEL
LIN {X 0,Y 656.744,Z 809.06,A -85,B 0,C 180,E1 5565.341,E2 5565.341} C_VEL
LIN {X 0,Y 656.887,Z 809.06,A -85,B 0,C 180,E1 5570.735,E2 5570.735} C_VEL
LIN {X 0,Y 657.022,Z 809.06,A -85,B 0,C 180,E1 5576.044,E2 5576.044} C_VEL
LIN {X 0,Y 657.232,Z 809.06,A -85,B 0,C 180,E1 5581.318,E2 5581.318} C_VEL
LIN {X 0,Y 656.887,Z 809.06,A -85,B 0,C 180,E1 5586.605,E2 5586.605} C_VEL
LIN {X 0,Y 656.843,Z 809.06,A -85,B 0,C 180,E1 5590.605,E2 5590.605} C_VEL
LIN {X 0,Y 656.789,Z 809.06,A -85,B 0,C 180,E1 5596.026,E2 5596.026} C_VEL
LIN {X 0,Y 656.675,Z 809.06,A -85,B 0,C 180,E1 5601.602,E2 5601.602} C_VEL
LIN {X 0,Y 656.554,Z 809.06,A -85,B 0,C 180,E1 5606.147,E2 5606.147} C_VEL
LIN {X 0,Y 656.542,Z 809.06,A -85,B 0,C 180,E1 5611.709,E2 5611.709} C_VEL
LIN {X 0,Y 652.541,Z 809.06,A -85,B 0,C 180,E1 5613.199,E2 5613.199} C_VEL
LIN {X 0,Y 648.553,Z 809.06,A -85,B 0,C 180,E1 5614.708,E2 5614.708} C_VEL
LIN {X 0,Y 648.484,Z 809.06,A -85,B 0,C 180,E1 5619.733,E2 5619.733} C_VEL
LIN {X 0,Y 648.645,Z 809.06,A -85,B 0,C 180,E1 5625.166,E2 5625.166} C_VEL
LIN {X 0,Y 648.659,Z 809.06,A -85,B 0,C 180,E1 5625.334,E2 5625.334} C_VEL
LIN {X 0,Y 651.222,Z 814.867,A -85,B 0,C 180,E1 5625.652,E2 5625.652} C_VEL
LIN {X 0,Y 674.551,Z 856.408,A -85,B 0,C 180,E1 5628.143,E2 5628.143} C_VEL
LIN {X 0,Y 673.288,Z 925.327,A -85,B 0,C 180,E1 5629.153,E2 5629.153} C_VEL
LIN {X 0,Y 671.037,Z 969.026,A -85,B 0,C 180,E1 5630.211,E2 5630.211} C_VEL
LIN {X 0,Y 668.285,Z 1013.712,A -85,B 0,C 180,E1 5631.815,E2 5631.815} C_VEL
LIN {X 0,Y 664.881,Z 1057.759,A -85,B 0,C 180,E1 5633.932,E2 5633.932} C_VEL
LIN {X 0,Y 661.279,Z 1100.163,A -85,B 0,C 180,E1 5636.55,E2 5636.55} C_VEL
LIN {X 0,Y 657.617,Z 1141.697,A -85,B 0,C 180,E1 5639.82,E2 5639.82} C_VEL
LIN {X 0,Y 654.674,Z 1176.943,A -85,B 0,C 180,E1 5643.279,E2 5643.279} C_VEL
LIN {X 0,Y 652.254,Z 1209.683,A -85,B 0,C 180,E1 5647.286,E2 5647.286} C_VEL
LIN {X 0,Y 650.636,Z 1235.774,A -85,B 0,C 180,E1 5651.348,E2 5651.348} C_VEL
LIN {X 0,Y 649.851,Z 1256.521,A -85,B 0,C 180,E1 5655.519,E2 5655.519} C_VEL
LIN {X 0,Y 649.415,Z 1270.403,A -85,B 0,C 180,E1 5659.267,E2 5659.267} C_VEL
LIN {X 0,Y 649.257,Z 1280.56,A -85,B 0,C 180,E1 5663.312,E2 5663.312} C_VEL
LIN {X 0,Y 649.202,Z 1285.871,A -85,B 0,C 180,E1 5667.326,E2 5667.326} C_VEL
LIN {X 0,Y 649.334,Z 1286.67,A -85,B 0,C 180,E1 5671.328,E2 5671.328} C_VEL
LIN {X 0,Y 649.193,Z 1282.919,A -85,B 0,C 180,E1 5675.337,E2 5675.337} C_VEL
LIN {X 0,Y 649.236,Z 1274.305,A -85,B 0,C 180,E1 5679.371,E2 5679.371} C_VEL
LIN {X 0,Y 649.706,Z 1260.73,A -85,B 0,C 180,E1 5683.443,E2 5683.443} C_VEL
LIN {X 0,Y 650.665,Z 1240.504,A -85,B 0,C 180,E1 5687.802,E2 5687.802} C_VEL
LIN {X 0,Y 652.1,Z 1214.292,A -85,B 0,C 180,E1 5692.051,E2 5692.051} C_VEL
LIN {X 0,Y 654.122,Z 1184.531,A -85,B 0,C 180,E1 5695.872,E2 5695.872} C_VEL
LIN {X 0,Y 657.114,Z 1147.943,A -85,B 0,C 180,E1 5699.623,E2 5699.623} C_VEL
LIN {X 0,Y 660.477,Z 1108.698,A -85,B 0,C 180,E1 5702.834,E2 5702.834} C_VEL
LIN {X 0,Y 664.199,Z 1065.637,A -85,B 0,C 180,E1 5705.639,E2 5705.639} C_VEL
LIN {X 0,Y 667.713,Z 1019.573,A -85,B 0,C 180,E1 5707.941,E2 5707.941} C_VEL
LIN {X 0,Y 670.774,Z 972.341,A -85,B 0,C 180,E1 5709.696,E2 5709.696} C_VEL
LIN {X 0,Y 673.123,Z 923.651,A -85,B 0,C 180,E1 5710.895,E2 5710.895} C_VEL
LIN {X 0,Y 674.287,Z 855.34,A -85,B 0,C 180,E1 5711.892,E2 5711.892} C_VEL
LIN {X 0,Y 650.355,Z 813.837,A -85,B 0,C 180,E1 5714.438,E2 5714.438} C_VEL
LIN {X 0,Y 648.675,Z 809.06,A -85,B 0,C 180,E1 5714.712,E2 5714.712} C_VEL
LIN {X 0,Y 648.489,Z 809.06,A -85,B 0,C 180,E1 5720.25,E2 5720.25} C_VEL
LIN {X 0,Y 648.537,Z 809.06,A -85,B 0,C 180,E1 5724.625,E2 5724.625} C_VEL
LIN {X 0,Y 648.536,Z 809.06,A -85,B 0,C 180,E1 5729.539,E2 5729.539} C_VEL
LIN {X 0,Y 648.58,Z 809.06,A -85,B 0,C 180,E1 5733.727,E2 5733.727} C_VEL
LIN {X 0,Y 648.573,Z 809.06,A -85,B 0,C 180,E1 5739.545,E2 5739.545} C_VEL
LIN {X 0,Y 648.532,Z 809.327,A -85,B 0,C 180,E1 5743.152,E2 5743.152} C_VEL
LIN {X 0,Y 667.981,Z 854.525,A -85,B 0,C 180,E1 5746.334,E2 5746.334} C_VEL
LIN {X 0,Y 668.313,Z 862.82,A -85,B 0,C 180,E1 5746.73,E2 5746.73} C_VEL
LIN {X 0,Y 664.695,Z 908.875,A -85,B 0,C 180,E1 5748.942,E2 5748.942} C_VEL
LIN {X 0,Y 661.031,Z 951.864,A -85,B 0,C 180,E1 5751.621,E2 5751.621} C_VEL
LIN {X 0,Y 657.532,Z 993.077,A -85,B 0,C 180,E1 5754.891,E2 5754.891} C_VEL
LIN {X 0,Y 654.495,Z 1029.46,A -85,B 0,C 180,E1 5758.511,E2 5758.511} C_VEL
LIN {X 0,Y 652.288,Z 1060.244,A -85,B 0,C 180,E1 5762.323,E2 5762.323} C_VEL
LIN {X 0,Y 650.624,Z 1085.945,A -85,B 0,C 180,E1 5766.333,E2 5766.333} C_VEL
LIN {X 0,Y 649.854,Z 1106.123,A -85,B 0,C 180,E1 5770.381,E2 5770.381} C_VEL
LIN {X 0,Y 649.321,Z 1121.194,A -85,B 0,C 180,E1 5774.486,E2 5774.486} C_VEL
LIN {X 0,Y 649.182,Z 1130.653,A -85,B 0,C 180,E1 5778.313,E2 5778.313} C_VEL
LIN {X 0,Y 648.933,Z 1135.597,A -85,B 0,C 180,E1 5781.872,E2 5781.872} C_VEL
LIN {X 0,Y 648.908,Z 1136.701,A -85,B 0,C 180,E1 5786.258,E2 5786.258} C_VEL
LIN {X 0,Y 649.204,Z 1132.089,A -85,B 0,C 180,E1 5790.799,E2 5790.799} C_VEL
LIN {X 0,Y 649.419,Z 1122.25,A -85,B 0,C 180,E1 5795.055,E2 5795.055} C_VEL
LIN {X 0,Y 649.835,Z 1107.57,A -85,B 0,C 180,E1 5799.195,E2 5799.195} C_VEL
LIN {X 0,Y 650.622,Z 1087.102,A -85,B 0,C 180,E1 5803.375,E2 5803.375} C_VEL
LIN {X 0,Y 652.198,Z 1060.828,A -85,B 0,C 180,E1 5807.511,E2 5807.511} C_VEL
LIN {X 0,Y 654.425,Z 1030.239,A -85,B 0,C 180,E1 5811.311,E2 5811.311} C_VEL
LIN {X 0,Y 657.268,Z 995.515,A -85,B 0,C 180,E1 5814.802,E2 5814.802} C_VEL
LIN {X 0,Y 660.726,Z 956.363,A -85,B 0,C 180,E1 5817.959,E2 5817.959} C_VEL
LIN {X 0,Y 664.295,Z 914.859,A -85,B 0,C 180,E1 5820.632,E2 5820.632} C_VEL
LIN {X 0,Y 667.676,Z 871.291,A -85,B 0,C 180,E1 5822.818,E2 5822.818} C_VEL
LIN {X 0,Y 668.464,Z 855.709,A -85,B 0,C 180,E1 5823.49,E2 5823.49} C_VEL
LIN {X 0,Y 652.399,Z 818.527,A -85,B 0,C 180,E1 5826.14,E2 5826.14} C_VEL
LIN {X 0,Y 648.508,Z 809.06,A -85,B 0,C 180,E1 5826.804,E2 5826.804} C_VEL
LIN {X 0,Y 648.531,Z 809.06,A -85,B 0,C 180,E1 5830.968,E2 5830.968} C_VEL
LIN {X 0,Y 648.727,Z 809.06,A -85,B 0,C 180,E1 5836.536,E2 5836.536} C_VEL
LIN {X 0,Y 649.024,Z 809.06,A -85,B 0,C 180,E1 5841.976,E2 5841.976} C_VEL
LIN {X 0,Y 649.151,Z 809.06,A -85,B 0,C 180,E1 5847.337,E2 5847.337} C_VEL
LIN {X 0,Y 649.002,Z 809.06,A -85,B 0,C 180,E1 5852.674,E2 5852.674} C_VEL
LIN {X 0,Y 648.96,Z 809.06,A -85,B 0,C 180,E1 5856.691,E2 5856.691} C_VEL
LIN {X 0,Y 648.937,Z 809.06,A -85,B 0,C 180,E1 5862.102,E2 5862.102} C_VEL
LIN {X 0,Y 648.922,Z 809.06,A -85,B 0,C 180,E1 5867.626,E2 5867.626} C_VEL
LIN {X 0,Y 648.707,Z 809.06,A -85,B 0,C 180,E1 5873.333,E2 5873.333} C_VEL
LIN {X 0,Y 648.66,Z 809.06,A -85,B 0,C 180,E1 5877.774,E2 5877.774} C_VEL
LIN {X 0,Y 648.609,Z 809.06,A -85,B 0,C 180,E1 5883.003,E2 5883.003} C_VEL
LIN {X 0,Y 648.493,Z 809.06,A -85,B 0,C 180,E1 5887.609,E2 5887.609} C_VEL
LIN {X 0,Y 648.591,Z 809.06,A -85,B 0,C 180,E1 5892.51,E2 5892.51} C_VEL
LIN {X 0,Y 648.49,Z 809.06,A -85,B 0,C 180,E1 5897.492,E2 5897.492} C_VEL
LIN {X 0,Y 648.471,Z 809.06,A -85,B 0,C 180,E1 5902.713,E2 5902.713} C_VEL
LIN {X 0,Y 648.496,Z 809.06,A -85,B 0,C 180,E1 5907.596,E2 5907.596} C_VEL
LIN {X 0,Y 648.75,Z 809.06,A -85,B 0,C 180,E1 5912.273,E2 5912.273} C_VEL
LIN {X 0,Y 648.762,Z 809.06,A -85,B 0,C 180,E1 5916.676,E2 5916.676} C_VEL
LIN {X 0,Y 648.868,Z 809.06,A -85,B 0,C 180,E1 5922.379,E2 5922.379} C_VEL
LIN {X 0,Y 648.892,Z 809.06,A -85,B 0,C 180,E1 5927.995,E2 5927.995} C_VEL
LIN {X 0,Y 649.066,Z 809.06,A -85,B 0,C 180,E1 5933.316,E2 5933.316} C_VEL
LIN {X 0,Y 649.08,Z 809.06,A -85,B 0,C 180,E1 5938.667,E2 5938.667} C_VEL
LIN {X 0,Y 649.091,Z 809.06,A -85,B 0,C 180,E1 5942.669,E2 5942.669} C_VEL
LIN {X 0,Y 649,Z 809.06,A -85,B 0,C 180,E1 5946.685,E2 5946.685} C_VEL
LIN {X 0,Y 648.9,Z 809.06,A -85,B 0,C 180,E1 5952.098,E2 5952.098} C_VEL
LIN {X 0,Y 648.876,Z 809.06,A -85,B 0,C 180,E1 5957.622,E2 5957.622} C_VEL
LIN {X 0,Y 648.697,Z 809.06,A -85,B 0,C 180,E1 5963.327,E2 5963.327} C_VEL
LIN {X 0,Y 648.597,Z 809.06,A -85,B 0,C 180,E1 5967.771,E2 5967.771} C_VEL
LIN {X 0,Y 648.588,Z 809.06,A -85,B 0,C 180,E1 5972.986,E2 5972.986} C_VEL
LIN {X 0,Y 648.553,Z 809.06,A -85,B 0,C 180,E1 5974.708,E2 5974.708} C_VEL
LIN {X 0,Y 647.276,Z 809.06,A -85,B 0,C 180,E1 5975.474,E2 5975.474} C_VEL
LIN {X 0,Y 640.656,Z 809.06,A -85,B 0,C 180,E1 5977.555,E2 5977.555} C_VEL
LIN {X 0,Y 640.582,Z 809.06,A -85,B 0,C 180,E1 5977.752,E2 5977.752} C_VEL
LIN {X 0,Y 640.715,Z 809.06,A -85,B 0,C 180,E1 5983.15,E2 5983.15} C_VEL
LIN {X 0,Y 640.759,Z 809.06,A -85,B 0,C 180,E1 5984.672,E2 5984.672} C_VEL
LIN {X 0,Y 643.264,Z 814.825,A -85,B 0,C 180,E1 5984.966,E2 5984.966} C_VEL
LIN {X 0,Y 668.445,Z 858.177,A -85,B 0,C 180,E1 5987.697,E2 5987.697} C_VEL
LIN {X 0,Y 667.215,Z 927.86,A -85,B 0,C 180,E1 5988.757,E2 5988.757} C_VEL
LIN {X 0,Y 664.738,Z 971.795,A -85,B 0,C 180,E1 5989.852,E2 5989.852} C_VEL
LIN {X 0,Y 661.613,Z 1017.452,A -85,B 0,C 180,E1 5991.543,E2 5991.543} C_VEL
LIN {X 0,Y 657.879,Z 1062.346,A -85,B 0,C 180,E1 5993.765,E2 5993.765} C_VEL
LIN {X 0,Y 654.079,Z 1103.672,A -85,B 0,C 180,E1 5996.41,E2 5996.41} C_VEL
LIN {X 0,Y 650.197,Z 1144.832,A -85,B 0,C 180,E1 5999.728,E2 5999.728} C_VEL
LIN {X 0,Y 646.967,Z 1180.428,A -85,B 0,C 180,E1 6003.34,E2 6003.34} C_VEL
LIN {X 0,Y 644.552,Z 1211.348,A -85,B 0,C 180,E1 6007.238,E2 6007.238} C_VEL
LIN {X 0,Y 642.798,Z 1237.866,A -85,B 0,C 180,E1 6011.492,E2 6011.492} C_VEL
LIN {X 0,Y 642.002,Z 1257.984,A -85,B 0,C 180,E1 6015.686,E2 6015.686} C_VEL
LIN {X 0,Y 641.507,Z 1272.344,A -85,B 0,C 180,E1 6019.819,E2 6019.819} C_VEL
LIN {X 0,Y 641.402,Z 1281.776,A -85,B 0,C 180,E1 6023.909,E2 6023.909} C_VEL
LIN {X 0,Y 641.298,Z 1285.871,A -85,B 0,C 180,E1 6027.293,E2 6027.293} C_VEL
LIN {X 0,Y 641.432,Z 1286.669,A -85,B 0,C 180,E1 6031.344,E2 6031.344} C_VEL
LIN {X 0,Y 641.296,Z 1282.919,A -85,B 0,C 180,E1 6035.403,E2 6035.403} C_VEL
LIN {X 0,Y 641.39,Z 1274.304,A -85,B 0,C 180,E1 6039.487,E2 6039.487} C_VEL
LIN {X 0,Y 641.865,Z 1260.731,A -85,B 0,C 180,E1 6043.61,E2 6043.61} C_VEL
LIN {X 0,Y 642.887,Z 1240.502,A -85,B 0,C 180,E1 6048.025,E2 6048.025} C_VEL
LIN {X 0,Y 644.453,Z 1214.294,A -85,B 0,C 180,E1 6052.326,E2 6052.326} C_VEL
LIN {X 0,Y 646.666,Z 1184.529,A -85,B 0,C 180,E1 6056.193,E2 6056.193} C_VEL
LIN {X 0,Y 649.898,Z 1147.936,A -85,B 0,C 180,E1 6059.986,E2 6059.986} C_VEL
LIN {X 0,Y 653.512,Z 1109.024,A -85,B 0,C 180,E1 6063.203,E2 6063.203} C_VEL
LIN {X 0,Y 657.539,Z 1065.921,A -85,B 0,C 180,E1 6066.038,E2 6066.038} C_VEL
LIN {X 0,Y 661.379,Z 1019.19,A -85,B 0,C 180,E1 6068.388,E2 6068.388} C_VEL
LIN {X 0,Y 664.647,Z 972.341,A -85,B 0,C 180,E1 6070.136,E2 6070.136} C_VEL
LIN {X 0,Y 667.204,Z 922.813,A -85,B 0,C 180,E1 6071.355,E2 6071.355} C_VEL
LIN {X 0,Y 668.098,Z 858.151,A -85,B 0,C 180,E1 6072.33,E2 6072.33} C_VEL
LIN {X 0,Y 643.046,Z 814.612,A -85,B 0,C 180,E1 6075.053,E2 6075.053} C_VEL
LIN {X 0,Y 640.73,Z 809.06,A -85,B 0,C 180,E1 6075.286,E2 6075.286} C_VEL
LIN {X 0,Y 640.564,Z 809.06,A -85,B 0,C 180,E1 6081.11,E2 6081.11} C_VEL
LIN {X 0,Y 640.587,Z 809.06,A -85,B 0,C 180,E1 6085.639,E2 6085.639} C_VEL
LIN {X 0,Y 640.625,Z 809.06,A -85,B 0,C 180,E1 6090.765,E2 6090.765} C_VEL
LIN {X 0,Y 640.614,Z 809.06,A -85,B 0,C 180,E1 6094.877,E2 6094.877} C_VEL
LIN {X 0,Y 640.631,Z 809.06,A -85,B 0,C 180,E1 6100.718,E2 6100.718} C_VEL
LIN {X 0,Y 640.628,Z 809.482,A -85,B 0,C 180,E1 6102.522,E2 6102.522} C_VEL
LIN {X 0,Y 660.074,Z 853.997,A -85,B 0,C 180,E1 6105.76,E2 6105.76} C_VEL
LIN {X 0,Y 662.15,Z 860.931,A -85,B 0,C 180,E1 6106.22,E2 6106.22} C_VEL
LIN {X 0,Y 658.273,Z 906.888,A -85,B 0,C 180,E1 6108.413,E2 6108.413} C_VEL
LIN {X 0,Y 654.332,Z 950.291,A -85,B 0,C 180,E1 6111.116,E2 6111.116} C_VEL
LIN {X 0,Y 650.558,Z 990.914,A -85,B 0,C 180,E1 6114.335,E2 6114.335} C_VEL
LIN {X 0,Y 647.249,Z 1027.751,A -85,B 0,C 180,E1 6117.993,E2 6117.993} C_VEL
LIN {X 0,Y 644.713,Z 1060.049,A -85,B 0,C 180,E1 6122.014,E2 6122.014} C_VEL
LIN {X 0,Y 642.928,Z 1085.774,A -85,B 0,C 180,E1 6126.07,E2 6126.07} C_VEL
LIN {X 0,Y 642.034,Z 1105.979,A -85,B 0,C 180,E1 6130.166,E2 6130.166} C_VEL
LIN {X 0,Y 641.444,Z 1121.081,A -85,B 0,C 180,E1 6134.32,E2 6134.32} C_VEL
LIN {X 0,Y 641.295,Z 1131.228,A -85,B 0,C 180,E1 6138.546,E2 6138.546} C_VEL
LIN {X 0,Y 640.989,Z 1135.844,A -85,B 0,C 180,E1 6142.158,E2 6142.158} C_VEL
LIN {X 0,Y 640.981,Z 1136.615,A -85,B 0,C 180,E1 6146.608,E2 6146.608} C_VEL
LIN {X 0,Y 641.237,Z 1132.993,A -85,B 0,C 180,E1 6150.29,E2 6150.29} C_VEL
LIN {X 0,Y 641.518,Z 1124.222,A -85,B 0,C 180,E1 6154.482,E2 6154.482} C_VEL
LIN {X 0,Y 641.947,Z 1110.34,A -85,B 0,C 180,E1 6158.667,E2 6158.667} C_VEL
LIN {X 0,Y 642.703,Z 1090.505,A -85,B 0,C 180,E1 6162.983,E2 6162.983} C_VEL
LIN {X 0,Y 644.315,Z 1065.189,A -85,B 0,C 180,E1 6167.156,E2 6167.156} C_VEL
LIN {X 0,Y 646.626,Z 1034.764,A -85,B 0,C 180,E1 6171.128,E2 6171.128} C_VEL
LIN {X 0,Y 649.873,Z 998.537,A -85,B 0,C 180,E1 6174.888,E2 6174.888} C_VEL
LIN {X 0,Y 653.511,Z 959.638,A -85,B 0,C 180,E1 6178.113,E2 6178.113} C_VEL
LIN {X 0,Y 657.393,Z 918.138,A -85,B 0,C 180,E1 6180.857,E2 6180.857} C_VEL
LIN {X 0,Y 660.983,Z 875.434,A -85,B 0,C 180,E1 6183.065,E2 6183.065} C_VEL
LIN {X 0,Y 661.696,Z 858.212,A -85,B 0,C 180,E1 6183.845,E2 6183.845} C_VEL
LIN {X 0,Y 645.755,Z 821.06,A -85,B 0,C 180,E1 6186.566,E2 6186.566} C_VEL
LIN {X 0,Y 640.6,Z 809.06,A -85,B 0,C 180,E1 6187.454,E2 6187.454} C_VEL
LIN {X 0,Y 640.552,Z 809.06,A -85,B 0,C 180,E1 6192.147,E2 6192.147} C_VEL
LIN {X 0,Y 640.801,Z 809.06,A -85,B 0,C 180,E1 6196.367,E2 6196.367} C_VEL
LIN {X 0,Y 641.063,Z 809.06,A -85,B 0,C 180,E1 6200.509,E2 6200.509} C_VEL
LIN {X 0,Y 641.178,Z 809.06,A -85,B 0,C 180,E1 6205.951,E2 6205.951} C_VEL
LIN {X 0,Y 641.299,Z 809.06,A -85,B 0,C 180,E1 6211.356,E2 6211.356} C_VEL
LIN {X 0,Y 641.052,Z 809.06,A -85,B 0,C 180,E1 6216.774,E2 6216.774} C_VEL
LIN {X 0,Y 641.005,Z 809.06,A -85,B 0,C 180,E1 6220.876,E2 6220.876} C_VEL
LIN {X 0,Y 641.012,Z 809.06,A -85,B 0,C 180,E1 6226.438,E2 6226.438} C_VEL
LIN {X 0,Y 640.81,Z 809.06,A -85,B 0,C 180,E1 6232.171,E2 6232.171} C_VEL
LIN {X 0,Y 640.749,Z 809.06,A -85,B 0,C 180,E1 6236.626,E2 6236.626} C_VEL
LIN {X 0,Y 640.656,Z 809.06,A -85,B 0,C 180,E1 6241.891,E2 6241.891} C_VEL
LIN {X 0,Y 640.582,Z 809.06,A -85,B 0,C 180,E1 6246.681,E2 6246.681} C_VEL
LIN {X 0,Y 640.616,Z 809.06,A -85,B 0,C 180,E1 6251.341,E2 6251.341} C_VEL
LIN {X 0,Y 640.584,Z 809.06,A -85,B 0,C 180,E1 6256.999,E2 6256.999} C_VEL
LIN {X 0,Y 640.562,Z 809.06,A -85,B 0,C 180,E1 6262.172,E2 6262.172} C_VEL
LIN {X 0,Y 640.595,Z 809.06,A -85,B 0,C 180,E1 6267.146,E2 6267.146} C_VEL
LIN {X 0,Y 640.78,Z 809.06,A -85,B 0,C 180,E1 6271.862,E2 6271.862} C_VEL
LIN {X 0,Y 640.845,Z 809.06,A -85,B 0,C 180,E1 6276.878,E2 6276.878} C_VEL
LIN {X 0,Y 640.94,Z 809.06,A -85,B 0,C 180,E1 6282.154,E2 6282.154} C_VEL
LIN {X 0,Y 640.956,Z 809.06,A -85,B 0,C 180,E1 6287.751,E2 6287.751} C_VEL
LIN {X 0,Y 641.154,Z 809.06,A -85,B 0,C 180,E1 6293.233,E2 6293.233} C_VEL
LIN {X 0,Y 641.181,Z 809.06,A -85,B 0,C 180,E1 6298.65,E2 6298.65} C_VEL
LIN {X 0,Y 641.189,Z 809.06,A -85,B 0,C 180,E1 6302.702,E2 6302.702} C_VEL
LIN {X 0,Y 641.11,Z 809.06,A -85,B 0,C 180,E1 6308.109,E2 6308.109} C_VEL
LIN {X 0,Y 640.956,Z 809.06,A -85,B 0,C 180,E1 6313.636,E2 6313.636} C_VEL
LIN {X 0,Y 640.942,Z 809.06,A -85,B 0,C 180,E1 6317.847,E2 6317.847} C_VEL
LIN {X 0,Y 640.786,Z 809.06,A -85,B 0,C 180,E1 6323.109,E2 6323.109} C_VEL
LIN {X 0,Y 640.658,Z 809.06,A -85,B 0,C 180,E1 6328.145,E2 6328.145} C_VEL
LIN {X 0,Y 640.686,Z 809.06,A -85,B 0,C 180,E1 6332.85,E2 6332.85} C_VEL
LIN {X 0,Y 640.582,Z 809.06,A -85,B 0,C 180,E1 6337.752,E2 6337.752} C_VEL
LIN {X 0,Y 638.099,Z 809.06,A -85,B 0,C 180,E1 6338.896,E2 6338.896} C_VEL
LIN {X 0,Y 632.703,Z 809.06,A -85,B 0,C 180,E1 6340.606,E2 6340.606} C_VEL
LIN {X 0,Y 632.605,Z 809.06,A -85,B 0,C 180,E1 6340.803,E2 6340.803} C_VEL
LIN {X 0,Y 632.839,Z 809.06,A -85,B 0,C 180,E1 6344.008,E2 6344.008} C_VEL
LIN {X 0,Y 635.338,Z 814.818,A -85,B 0,C 180,E1 6344.329,E2 6344.329} C_VEL
LIN {X 0,Y 662.741,Z 861.884,A -85,B 0,C 180,E1 6347.301,E2 6347.301} C_VEL
LIN {X 0,Y 661.264,Z 927.835,A -85,B 0,C 180,E1 6348.304,E2 6348.304} C_VEL
LIN {X 0,Y 658.608,Z 972.322,A -85,B 0,C 180,E1 6349.419,E2 6349.419} C_VEL
LIN {X 0,Y 655.383,Z 1016.779,A -85,B 0,C 180,E1 6351.075,E2 6351.075} C_VEL
LIN {X 0,Y 651.424,Z 1061.441,A -85,B 0,C 180,E1 6353.292,E2 6353.292} C_VEL
LIN {X 0,Y 647.356,Z 1102.545,A -85,B 0,C 180,E1 6355.924,E2 6355.924} C_VEL
LIN {X 0,Y 643.076,Z 1144.684,A -85,B 0,C 180,E1 6359.343,E2 6359.343} C_VEL
LIN {X 0,Y 639.539,Z 1180.721,A -85,B 0,C 180,E1 6363.041,E2 6363.041} C_VEL
LIN {X 0,Y 636.918,Z 1211.35,A -85,B 0,C 180,E1 6366.949,E2 6366.949} C_VEL
LIN {X 0,Y 635.124,Z 1235.91,A -85,B 0,C 180,E1 6370.899,E2 6370.899} C_VEL
LIN {X 0,Y 634.161,Z 1254.989,A -85,B 0,C 180,E1 6374.799,E2 6374.799} C_VEL
LIN {X 0,Y 633.634,Z 1270.403,A -85,B 0,C 180,E1 6378.996,E2 6378.996} C_VEL
LIN {X 0,Y 633.448,Z 1280.56,A -85,B 0,C 180,E1 6383.144,E2 6383.144} C_VEL
LIN {X 0,Y 633.417,Z 1285.871,A -85,B 0,C 180,E1 6387.26,E2 6387.26} C_VEL
LIN {X 0,Y 633.553,Z 1286.669,A -85,B 0,C 180,E1 6391.361,E2 6391.361} C_VEL
LIN {X 0,Y 633.399,Z 1282.919,A -85,B 0,C 180,E1 6395.47,E2 6395.47} C_VEL
LIN {X 0,Y 633.514,Z 1274.304,A -85,B 0,C 180,E1 6399.606,E2 6399.606} C_VEL
LIN {X 0,Y 634.052,Z 1260.732,A -85,B 0,C 180,E1 6403.781,E2 6403.781} C_VEL
LIN {X 0,Y 635.064,Z 1241.753,A -85,B 0,C 180,E1 6408.012,E2 6408.012} C_VEL
LIN {X 0,Y 636.696,Z 1216.297,A -85,B 0,C 180,E1 6412.31,E2 6412.31} C_VEL
LIN {X 0,Y 639.071,Z 1186.591,A -85,B 0,C 180,E1 6416.284,E2 6416.284} C_VEL
LIN {X 0,Y 642.512,Z 1150.253,A -85,B 0,C 180,E1 6420.131,E2 6420.131} C_VEL
LIN {X 0,Y 646.34,Z 1112.085,A -85,B 0,C 180,E1 6423.375,E2 6423.375} C_VEL
LIN {X 0,Y 650.691,Z 1068.211,A -85,B 0,C 180,E1 6426.323,E2 6426.323} C_VEL
LIN {X 0,Y 654.748,Z 1023,A -85,B 0,C 180,E1 6428.66,E2 6428.66} C_VEL
LIN {X 0,Y 658.465,Z 973.476,A -85,B 0,C 180,E1 6430.548,E2 6430.548} C_VEL
LIN {X 0,Y 661.156,Z 925.119,A -85,B 0,C 180,E1 6431.765,E2 6431.765} C_VEL
LIN {X 0,Y 662.276,Z 861.256,A -85,B 0,C 180,E1 6432.746,E2 6432.746} C_VEL
LIN {X 0,Y 638.503,Z 820.602,A -85,B 0,C 180,E1 6435.27,E2 6435.27} C_VEL
LIN {X 0,Y 632.951,Z 810.531,A -85,B 0,C 180,E1 6435.761,E2 6435.761} C_VEL
LIN {X 0,Y 632.794,Z 809.06,A -85,B 0,C 180,E1 6435.792,E2 6435.792} C_VEL
LIN {X 0,Y 632.665,Z 809.06,A -85,B 0,C 180,E1 6442.005,E2 6442.005} C_VEL
LIN {X 0,Y 632.627,Z 809.06,A -85,B 0,C 180,E1 6446.708,E2 6446.708} C_VEL
LIN {X 0,Y 632.683,Z 809.06,A -85,B 0,C 180,E1 6452.077,E2 6452.077} C_VEL
LIN {X 0,Y 632.66,Z 809.06,A -85,B 0,C 180,E1 6457.534,E2 6457.534} C_VEL
LIN {X 0,Y 632.712,Z 809.586,A -85,B 0,C 180,E1 6461.868,E2 6461.868} C_VEL
LIN {X 0,Y 652.597,Z 854.495,A -85,B 0,C 180,E1 6465.244,E2 6465.244} C_VEL
LIN {X 0,Y 655.651,Z 863.699,A -85,B 0,C 180,E1 6465.896,E2 6465.896} C_VEL
LIN {X 0,Y 651.492,Z 909.336,A -85,B 0,C 180,E1 6468.121,E2 6468.121} C_VEL
LIN {X 0,Y 647.315,Z 952.264,A -85,B 0,C 180,E1 6470.849,E2 6470.849} C_VEL
LIN {X 0,Y 643.13,Z 994.382,A -85,B 0,C 180,E1 6474.269,E2 6474.269} C_VEL
LIN {X 0,Y 639.629,Z 1030.499,A -85,B 0,C 180,E1 6477.969,E2 6477.969} C_VEL
LIN {X 0,Y 637.036,Z 1061.056,A -85,B 0,C 180,E1 6481.868,E2 6481.868} C_VEL
LIN {X 0,Y 635.044,Z 1087.524,A -85,B 0,C 180,E1 6486.146,E2 6486.146} C_VEL
LIN {X 0,Y 634.162,Z 1107.313,A -85,B 0,C 180,E1 6490.293,E2 6490.293} C_VEL
LIN {X 0,Y 633.55,Z 1121.868,A -85,B 0,C 180,E1 6494.459,E2 6494.459} C_VEL
LIN {X 0,Y 633.373,Z 1131.801,A -85,B 0,C 180,E1 6498.787,E2 6498.787} C_VEL
LIN {X 0,Y 633.071,Z 1136.09,A -85,B 0,C 180,E1 6502.45,E2 6502.45} C_VEL
LIN {X 0,Y 633.033,Z 1136.906,A -85,B 0,C 180,E1 6505.444,E2 6505.444} C_VEL
LIN {X 0,Y 633.133,Z 1135.252,A -85,B 0,C 180,E1 6508.509,E2 6508.509} C_VEL
LIN {X 0,Y 633.394,Z 1129.35,A -85,B 0,C 180,E1 6512.436,E2 6512.436} C_VEL
LIN {X 0,Y 633.671,Z 1118.369,A -85,B 0,C 180,E1 6516.592,E2 6516.592} C_VEL
LIN {X 0,Y 634.278,Z 1102.85,A -85,B 0,C 180,E1 6520.649,E2 6520.649} C_VEL
LIN {X 0,Y 635.62,Z 1080.883,A -85,B 0,C 180,E1 6524.949,E2 6524.949} C_VEL
LIN {X 0,Y 637.793,Z 1051.948,A -85,B 0,C 180,E1 6529.297,E2 6529.297} C_VEL
LIN {X 0,Y 640.56,Z 1020.204,A -85,B 0,C 180,E1 6533.083,E2 6533.083} C_VEL
LIN {X 0,Y 644.223,Z 982.594,A -85,B 0,C 180,E1 6536.683,E2 6536.683} C_VEL
LIN {X 0,Y 648.36,Z 942.138,A -85,B 0,C 180,E1 6539.759,E2 6539.759} C_VEL
LIN {X 0,Y 652.602,Z 897.745,A -85,B 0,C 180,E1 6542.42,E2 6542.42} C_VEL
LIN {X 0,Y 655.432,Z 861.925,A -85,B 0,C 180,E1 6544.117,E2 6544.117} C_VEL
LIN {X 0,Y 639.575,Z 824.432,A -85,B 0,C 180,E1 6546.926,E2 6546.926} C_VEL
LIN {X 0,Y 632.678,Z 809.06,A -85,B 0,C 180,E1 6548.111,E2 6548.111} C_VEL
LIN {X 0,Y 632.669,Z 809.06,A -85,B 0,C 180,E1 6553.351,E2 6553.351} C_VEL
LIN {X 0,Y 633.103,Z 809.06,A -85,B 0,C 180,E1 6558.998,E2 6558.998} C_VEL
LIN {X 0,Y 633.226,Z 809.06,A -85,B 0,C 180,E1 6564.528,E2 6564.528} C_VEL
LIN {X 0,Y 633.233,Z 809.06,A -85,B 0,C 180,E1 6568.638,E2 6568.638} C_VEL
LIN {X 0,Y 633.209,Z 809.06,A -85,B 0,C 180,E1 6572.741,E2 6572.741} C_VEL
LIN {X 0,Y 633.205,Z 809.06,A -85,B 0,C 180,E1 6578.238,E2 6578.238} C_VEL
LIN {X 0,Y 633.09,Z 809.06,A -85,B 0,C 180,E1 6583.814,E2 6583.814} C_VEL
LIN {X 0,Y 633.055,Z 809.06,A -85,B 0,C 180,E1 6588.083,E2 6588.083} C_VEL
LIN {X 0,Y 632.886,Z 809.06,A -85,B 0,C 180,E1 6592.464,E2 6592.464} C_VEL
LIN {X 0,Y 632.804,Z 809.06,A -85,B 0,C 180,E1 6597.937,E2 6597.937} C_VEL
LIN {X 0,Y 632.763,Z 809.06,A -85,B 0,C 180,E1 6603.322,E2 6603.322} C_VEL
LIN {X 0,Y 632.652,Z 809.06,A -85,B 0,C 180,E1 6608.396,E2 6608.396} C_VEL
LIN {X 0,Y 632.705,Z 809.06,A -85,B 0,C 180,E1 6614.239,E2 6614.239} C_VEL
LIN {X 0,Y 632.655,Z 809.06,A -85,B 0,C 180,E1 6619.853,E2 6619.853} C_VEL
LIN {X 0,Y 632.62,Z 809.06,A -85,B 0,C 180,E1 6625.025,E2 6625.025} C_VEL
LIN {X 0,Y 632.747,Z 809.06,A -85,B 0,C 180,E1 6629.903,E2 6629.903} C_VEL
LIN {X 0,Y 632.915,Z 809.06,A -85,B 0,C 180,E1 6635.138,E2 6635.138} C_VEL
LIN {X 0,Y 633.022,Z 809.06,A -85,B 0,C 180,E1 6640.478,E2 6640.478} C_VEL
LIN {X 0,Y 633.012,Z 809.06,A -85,B 0,C 180,E1 6644.778,E2 6644.778} C_VEL
LIN {X 0,Y 633.146,Z 809.06,A -85,B 0,C 180,E1 6650.384,E2 6650.384} C_VEL
LIN {X 0,Y 633.326,Z 809.06,A -85,B 0,C 180,E1 6655.896,E2 6655.896} C_VEL
LIN {X 0,Y 633.55,Z 809.06,A -85,B 0,C 180,E1 6661.367,E2 6661.367} C_VEL
LIN {X 0,Y 633.185,Z 809.06,A -85,B 0,C 180,E1 6666.853,E2 6666.853} C_VEL
LIN {X 0,Y 633.085,Z 809.06,A -85,B 0,C 180,E1 6672.405,E2 6672.405} C_VEL
LIN {X 0,Y 633.029,Z 809.06,A -85,B 0,C 180,E1 6678.078,E2 6678.078} C_VEL
LIN {X 0,Y 632.89,Z 809.06,A -85,B 0,C 180,E1 6682.458,E2 6682.458} C_VEL
LIN {X 0,Y 632.738,Z 809.06,A -85,B 0,C 180,E1 6687.909,E2 6687.909} C_VEL
LIN {X 0,Y 632.759,Z 809.06,A -85,B 0,C 180,E1 6693.315,E2 6693.315} C_VEL
LIN {X 0,Y 632.673,Z 809.06,A -85,B 0,C 180,E1 6698.386,E2 6698.386} C_VEL
LIN {X 0,Y 632.605,Z 809.06,A -85,B 0,C 180,E1 6700.803,E2 6700.803} C_VEL
LIN {X 0,Y 628.714,Z 809.06,A -85,B 0,C 180,E1 6701.817,E2 6701.817} C_VEL
LIN {X 0,Y 624.794,Z 809.06,A -85,B 0,C 180,E1 6702.842,E2 6702.842} C_VEL
LIN {X 0,Y 624.856,Z 809.523,A -85,B 0,C 180,E1 6703.366,E2 6703.366} C_VEL
LIN {X 0,Y 630.227,Z 819.837,A -85,B 0,C 180,E1 6703.983,E2 6703.983} C_VEL
LIN {X 0,Y 656.786,Z 864.876,A -85,B 0,C 180,E1 6706.863,E2 6706.863} C_VEL
LIN {X 0,Y 655.33,Z 928.668,A -85,B 0,C 180,E1 6707.859,E2 6707.859} C_VEL
LIN {X 0,Y 652.556,Z 972.322,A -85,B 0,C 180,E1 6708.963,E2 6708.963} C_VEL
LIN {X 0,Y 649.205,Z 1015.624,A -85,B 0,C 180,E1 6710.575,E2 6710.575} C_VEL
LIN {X 0,Y 645.015,Z 1060.313,A -85,B 0,C 180,E1 6712.795,E2 6712.795} C_VEL
LIN {X 0,Y 640.671,Z 1101.533,A -85,B 0,C 180,E1 6715.436,E2 6715.436} C_VEL
LIN {X 0,Y 636.185,Z 1142.467,A -85,B 0,C 180,E1 6718.764,E2 6718.764} C_VEL
LIN {X 0,Y 632.425,Z 1177.831,A -85,B 0,C 180,E1 6722.365,E2 6722.365} C_VEL
LIN {X 0,Y 629.473,Z 1210.087,A -85,B 0,C 180,E1 6726.473,E2 6726.473} C_VEL
LIN {X 0,Y 627.408,Z 1235.911,A -85,B 0,C 180,E1 6730.655,E2 6730.655} C_VEL
LIN {X 0,Y 626.308,Z 1255.828,A -85,B 0,C 180,E1 6734.801,E2 6734.801} C_VEL
LIN {X 0,Y 625.772,Z 1270.403,A -85,B 0,C 180,E1 6738.856,E2 6738.856} C_VEL
LIN {X 0,Y 625.548,Z 1280.56,A -85,B 0,C 180,E1 6743.057,E2 6743.057} C_VEL
LIN {X 0,Y 625.512,Z 1285.872,A -85,B 0,C 180,E1 6747.225,E2 6747.225} C_VEL
LIN {X 0,Y 625.65,Z 1286.669,A -85,B 0,C 180,E1 6751.378,E2 6751.378} C_VEL
LIN {X 0,Y 625.504,Z 1282.919,A -85,B 0,C 180,E1 6755.539,E2 6755.539} C_VEL
LIN {X 0,Y 625.641,Z 1274.304,A -85,B 0,C 180,E1 6759.728,E2 6759.728} C_VEL
LIN {X 0,Y 626.217,Z 1260.734,A -85,B 0,C 180,E1 6763.957,E2 6763.957} C_VEL
LIN {X 0,Y 627.291,Z 1241.755,A -85,B 0,C 180,E1 6768.243,E2 6768.243} C_VEL
LIN {X 0,Y 629.061,Z 1216.295,A -85,B 0,C 180,E1 6772.596,E2 6772.596} C_VEL
LIN {X 0,Y 631.678,Z 1186.587,A -85,B 0,C 180,E1 6776.616,E2 6776.616} C_VEL
LIN {X 0,Y 635.287,Z 1150.811,A -85,B 0,C 180,E1 6780.453,E2 6780.453} C_VEL
LIN {X 0,Y 639.441,Z 1112.244,A -85,B 0,C 180,E1 6783.77,E2 6783.77} C_VEL
LIN {X 0,Y 644.023,Z 1069.206,A -85,B 0,C 180,E1 6786.692,E2 6786.692} C_VEL
LIN {X 0,Y 648.343,Z 1024.156,A -85,B 0,C 180,E1 6789.056,E2 6789.056} C_VEL
LIN {X 0,Y 652.308,Z 974.535,A -85,B 0,C 180,E1 6790.97,E2 6790.97} C_VEL
LIN {X 0,Y 655.171,Z 926.857,A -85,B 0,C 180,E1 6792.194,E2 6792.194} C_VEL
LIN {X 0,Y 656.463,Z 864.611,A -85,B 0,C 180,E1 6793.167,E2 6793.167} C_VEL
LIN {X 0,Y 637.256,Z 831.55,A -85,B 0,C 180,E1 6795.204,E2 6795.204} C_VEL
LIN {X 0,Y 627.503,Z 815.791,A -85,B 0,C 180,E1 6796.048,E2 6796.048} C_VEL
LIN {X 0,Y 624.818,Z 809.06,A -85,B 0,C 180,E1 6796.361,E2 6796.361} C_VEL
LIN {X 0,Y 624.685,Z 809.06,A -85,B 0,C 180,E1 6801.031,E2 6801.031} C_VEL
LIN {X 0,Y 624.672,Z 809.06,A -85,B 0,C 180,E1 6806.197,E2 6806.197} C_VEL
LIN {X 0,Y 624.732,Z 809.06,A -85,B 0,C 180,E1 6811.071,E2 6811.071} C_VEL
LIN {X 0,Y 624.755,Z 809.06,A -85,B 0,C 180,E1 6815.722,E2 6815.722} C_VEL
LIN {X 0,Y 624.828,Z 809.677,A -85,B 0,C 180,E1 6821.224,E2 6821.224} C_VEL
LIN {X 0,Y 644.406,Z 853.035,A -85,B 0,C 180,E1 6824.57,E2 6824.57} C_VEL
LIN {X 0,Y 649.128,Z 866.452,A -85,B 0,C 180,E1 6825.562,E2 6825.562} C_VEL
LIN {X 0,Y 644.616,Z 913.24,A -85,B 0,C 180,E1 6827.907,E2 6827.907} C_VEL
LIN {X 0,Y 639.901,Z 957.595,A -85,B 0,C 180,E1 6830.828,E2 6830.828} C_VEL
LIN {X 0,Y 635.867,Z 995.894,A -85,B 0,C 180,E1 6834.032,E2 6834.032} C_VEL
LIN {X 0,Y 632.147,Z 1031.742,A -85,B 0,C 180,E1 6837.773,E2 6837.773} C_VEL
LIN {X 0,Y 629.371,Z 1062.062,A -85,B 0,C 180,E1 6841.719,E2 6841.719} C_VEL
LIN {X 0,Y 627.347,Z 1087.355,A -85,B 0,C 180,E1 6845.875,E2 6845.875} C_VEL
LIN {X 0,Y 626.324,Z 1107.173,A -85,B 0,C 180,E1 6850.073,E2 6850.073} C_VEL
LIN {X 0,Y 625.672,Z 1122.307,A -85,B 0,C 180,E1 6854.484,E2 6854.484} C_VEL
LIN {X 0,Y 625.48,Z 1131.082,A -85,B 0,C 180,E1 6858.303,E2 6858.303} C_VEL
LIN {X 0,Y 625.124,Z 1136.315,A -85,B 0,C 180,E1 6862.751,E2 6862.751} C_VEL
LIN {X 0,Y 625.163,Z 1136.205,A -85,B 0,C 180,E1 6867.336,E2 6867.336} C_VEL
LIN {X 0,Y 625.46,Z 1131.714,A -85,B 0,C 180,E1 6871.253,E2 6871.253} C_VEL
LIN {X 0,Y 625.766,Z 1122.33,A -85,B 0,C 180,E1 6875.415,E2 6875.415} C_VEL
LIN {X 0,Y 626.282,Z 1107.665,A -85,B 0,C 180,E1 6879.718,E2 6879.718} C_VEL
LIN {X 0,Y 627.348,Z 1087.659,A -85,B 0,C 180,E1 6883.983,E2 6883.983} C_VEL
LIN {X 0,Y 629.439,Z 1060.792,A -85,B 0,C 180,E1 6888.379,E2 6888.379} C_VEL
LIN {X 0,Y 632.307,Z 1029.344,A -85,B 0,C 180,E1 6892.416,E2 6892.416} C_VEL
LIN {X 0,Y 636.022,Z 993.922,A -85,B 0,C 180,E1 6896.061,E2 6896.061} C_VEL
LIN {X 0,Y 640.372,Z 953.984,A -85,B 0,C 180,E1 6899.342,E2 6899.342} C_VEL
LIN {X 0,Y 644.836,Z 912.155,A -85,B 0,C 180,E1 6902.059,E2 6902.059} C_VEL
LIN {X 0,Y 648.855,Z 869.842,A -85,B 0,C 180,E1 6904.196,E2 6904.196} C_VEL
LIN {X 0,Y 648.797,Z 864.69,A -85,B 0,C 180,E1 6904.464,E2 6904.464} C_VEL
LIN {X 0,Y 633.824,Z 828.982,A -85,B 0,C 180,E1 6907.213,E2 6907.213} C_VEL
LIN {X 0,Y 624.823,Z 809.06,A -85,B 0,C 180,E1 6908.737,E2 6908.737} C_VEL
LIN {X 0,Y 624.892,Z 809.06,A -85,B 0,C 180,E1 6914.58,E2 6914.58} C_VEL
LIN {X 0,Y 625.258,Z 809.06,A -85,B 0,C 180,E1 6920.266,E2 6920.266} C_VEL
LIN {X 0,Y 625.371,Z 809.06,A -85,B 0,C 180,E1 6925.849,E2 6925.849} C_VEL
LIN {X 0,Y 625.488,Z 809.06,A -85,B 0,C 180,E1 6931.39,E2 6931.39} C_VEL
LIN {X 0,Y 625.239,Z 809.06,A -85,B 0,C 180,E1 6936.946,E2 6936.946} C_VEL
LIN {X 0,Y 625.185,Z 809.06,A -85,B 0,C 180,E1 6941.154,E2 6941.154} C_VEL
LIN {X 0,Y 625.169,Z 809.06,A -85,B 0,C 180,E1 6946.866,E2 6946.866} C_VEL
LIN {X 0,Y 625.028,Z 809.06,A -85,B 0,C 180,E1 6951.268,E2 6951.268} C_VEL
LIN {X 0,Y 624.868,Z 809.06,A -85,B 0,C 180,E1 6956.532,E2 6956.532} C_VEL
LIN {X 0,Y 624.851,Z 809.06,A -85,B 0,C 180,E1 6962.184,E2 6962.184} C_VEL
LIN {X 0,Y 624.768,Z 809.06,A -85,B 0,C 180,E1 6967.21,E2 6967.21} C_VEL
LIN {X 0,Y 624.767,Z 809.06,A -85,B 0,C 180,E1 6972.633,E2 6972.633} C_VEL
LIN {X 0,Y 624.698,Z 809.06,A -85,B 0,C 180,E1 6977.372,E2 6977.372} C_VEL
LIN {X 0,Y 624.728,Z 809.06,A -85,B 0,C 180,E1 6982.966,E2 6982.966} C_VEL
LIN {X 0,Y 624.759,Z 809.06,A -85,B 0,C 180,E1 6987.855,E2 6987.855} C_VEL
LIN {X 0,Y 624.955,Z 809.06,A -85,B 0,C 180,E1 6993.47,E2 6993.47} C_VEL
LIN {X 0,Y 625.063,Z 809.06,A -85,B 0,C 180,E1 6998.741,E2 6998.741} C_VEL
LIN {X 0,Y 625.133,Z 809.06,A -85,B 0,C 180,E1 7003.14,E2 7003.14} C_VEL
LIN {X 0,Y 625.204,Z 809.06,A -85,B 0,C 180,E1 7008.853,E2 7008.853} C_VEL
LIN {X 0,Y 625.32,Z 809.06,A -85,B 0,C 180,E1 7013.14,E2 7013.14} C_VEL
LIN {X 0,Y 625.384,Z 809.06,A -85,B 0,C 180,E1 7018.616,E2 7018.616} C_VEL
LIN {X 0,Y 625.395,Z 809.06,A -85,B 0,C 180,E1 7022.77,E2 7022.77} C_VEL
LIN {X 0,Y 625.285,Z 809.06,A -85,B 0,C 180,E1 7028.337,E2 7028.337} C_VEL
LIN {X 0,Y 625.145,Z 809.06,A -85,B 0,C 180,E1 7033.988,E2 7033.988} C_VEL
LIN {X 0,Y 625.093,Z 809.06,A -85,B 0,C 180,E1 7039.464,E2 7039.464} C_VEL
LIN {X 0,Y 624.915,Z 809.06,A -85,B 0,C 180,E1 7044.271,E2 7044.271} C_VEL
LIN {X 0,Y 624.801,Z 809.06,A -85,B 0,C 180,E1 7049.456,E2 7049.456} C_VEL
LIN {X 0,Y 624.775,Z 809.06,A -85,B 0,C 180,E1 7054.674,E2 7054.674} C_VEL
LIN {X 0,Y 624.693,Z 809.06,A -85,B 0,C 180,E1 7059.273,E2 7059.273} C_VEL
LIN {X 0,Y 624.794,Z 809.06,A -85,B 0,C 180,E1 7062.842,E2 7062.842} C_VEL
LIN {X 0,Y 625.818,Z 812.093,A -85,B 0,C 180,E1 7063.391,E2 7063.391} C_VEL
LIN {X 0,Y 628.218,Z 820.206,A -85,B 0,C 180,E1 7063.82,E2 7063.82} C_VEL
LIN {X 0,Y 632.283,Z 835.847,A -85,B 0,C 180,E1 7064.393,E2 7064.393} C_VEL
LIN {X 0,Y 633.28,Z 837.737,A -85,B 0,C 180,E1 7064.503,E2 7064.503} C_VEL
LIN {X 0,Y 651.016,Z 868.154,A -85,B 0,C 180,E1 7066.434,E2 7066.434} C_VEL
LIN {X 0,Y 649.378,Z 930.416,A -85,B 0,C 180,E1 7067.423,E2 7067.423} C_VEL
LIN {X 0,Y 646.346,Z 974.453,A -85,B 0,C 180,E1 7068.566,E2 7068.566} C_VEL
LIN {X 0,Y 642.612,Z 1019.458,A -85,B 0,C 180,E1 7070.287,E2 7070.287} C_VEL
LIN {X 0,Y 638.156,Z 1064.006,A -85,B 0,C 180,E1 7072.561,E2 7072.561} C_VEL
LIN {X 0,Y 633.491,Z 1104.904,A -85,B 0,C 180,E1 7075.266,E2 7075.266} C_VEL
LIN {X 0,Y 628.78,Z 1145.701,A -85,B 0,C 180,E1 7078.666,E2 7078.666} C_VEL
LIN {X 0,Y 624.718,Z 1181.417,A -85,B 0,C 180,E1 7082.433,E2 7082.433} C_VEL
LIN {X 0,Y 621.805,Z 1211.354,A -85,B 0,C 180,E1 7086.355,E2 7086.355} C_VEL
LIN {X 0,Y 619.548,Z 1237.862,A -85,B 0,C 180,E1 7090.77,E2 7090.77} C_VEL
LIN {X 0,Y 618.421,Z 1257.5,A -85,B 0,C 180,E1 7095,E2 7095} C_VEL
LIN {X 0,Y 617.853,Z 1272.345,A -85,B 0,C 180,E1 7099.425,E2 7099.425} C_VEL
LIN {X 0,Y 617.73,Z 1281.767,A -85,B 0,C 180,E1 7103.675,E2 7103.675} C_VEL
LIN {X 0,Y 617.635,Z 1285.872,A -85,B 0,C 180,E1 7107.19,E2 7107.19} C_VEL
LIN {X 0,Y 617.769,Z 1286.669,A -85,B 0,C 180,E1 7111.396,E2 7111.396} C_VEL
LIN {X 0,Y 617.61,Z 1282.919,A -85,B 0,C 180,E1 7115.61,E2 7115.61} C_VEL
LIN {X 0,Y 617.768,Z 1274.303,A -85,B 0,C 180,E1 7119.853,E2 7119.853} C_VEL
LIN {X 0,Y 618.389,Z 1260.735,A -85,B 0,C 180,E1 7124.138,E2 7124.138} C_VEL
LIN {X 0,Y 619.507,Z 1241.756,A -85,B 0,C 180,E1 7128.481,E2 7128.481} C_VEL
LIN {X 0,Y 621.425,Z 1216.292,A -85,B 0,C 180,E1 7132.889,E2 7132.889} C_VEL
LIN {X 0,Y 624.391,Z 1185.643,A -85,B 0,C 180,E1 7137.066,E2 7137.066} C_VEL
LIN {X 0,Y 628.442,Z 1148.619,A -85,B 0,C 180,E1 7141.05,E2 7141.05} C_VEL
LIN {X 0,Y 632.769,Z 1111.181,A -85,B 0,C 180,E1 7144.263,E2 7144.263} C_VEL
LIN {X 0,Y 637.605,Z 1068.383,A -85,B 0,C 180,E1 7147.18,E2 7147.18} C_VEL
LIN {X 0,Y 642.072,Z 1024.484,A -85,B 0,C 180,E1 7149.495,E2 7149.495} C_VEL
LIN {X 0,Y 646.257,Z 974.979,A -85,B 0,C 180,E1 7151.42,E2 7151.42} C_VEL
LIN {X 0,Y 649.326,Z 926.832,A -85,B 0,C 180,E1 7152.664,E2 7152.664} C_VEL
LIN {X 0,Y 650.701,Z 867.836,A -85,B 0,C 180,E1 7153.597,E2 7153.597} C_VEL
LIN {X 0,Y 635.261,Z 841.462,A -85,B 0,C 180,E1 7155.199,E2 7155.199} C_VEL
LIN {X 0,Y 622.194,Z 820.813,A -85,B 0,C 180,E1 7156.335,E2 7156.335} C_VEL
LIN {X 0,Y 616.862,Z 809.06,A -85,B 0,C 180,E1 7156.938,E2 7156.938} C_VEL
LIN {X 0,Y 616.756,Z 809.06,A -85,B 0,C 180,E1 7162.231,E2 7162.231} C_VEL
LIN {X 0,Y 616.756,Z 809.06,A -85,B 0,C 180,E1 7167.385,E2 7167.385} C_VEL
LIN {X 0,Y 616.824,Z 809.06,A -85,B 0,C 180,E1 7172.261,E2 7172.261} C_VEL
LIN {X 0,Y 616.818,Z 809.06,A -85,B 0,C 180,E1 7176.924,E2 7176.924} C_VEL
LIN {X 0,Y 616.985,Z 809.06,A -85,B 0,C 180,E1 7180.569,E2 7180.569} C_VEL
LIN {X 0,Y 623.553,Z 823.987,A -85,B 0,C 180,E1 7181.638,E2 7181.638} C_VEL
LIN {X 0,Y 639.716,Z 860.792,A -85,B 0,C 180,E1 7184.584,E2 7184.584} C_VEL
LIN {X 0,Y 642.599,Z 870.145,A -85,B 0,C 180,E1 7185.266,E2 7185.266} C_VEL
LIN {X 0,Y 637.735,Z 917.018,A -85,B 0,C 180,E1 7187.687,E2 7187.687} C_VEL
LIN {X 0,Y 632.892,Z 959.458,A -85,B 0,C 180,E1 7190.552,E2 7190.552} C_VEL
LIN {X 0,Y 628.604,Z 997.41,A -85,B 0,C 180,E1 7193.79,E2 7193.79} C_VEL
LIN {X 0,Y 624.662,Z 1032.988,A -85,B 0,C 180,E1 7197.573,E2 7197.573} C_VEL
LIN {X 0,Y 621.592,Z 1064.208,A -85,B 0,C 180,E1 7201.741,E2 7201.741} C_VEL
LIN {X 0,Y 619.477,Z 1089.102,A -85,B 0,C 180,E1 7205.95,E2 7205.95} C_VEL
LIN {X 0,Y 618.454,Z 1108.442,A -85,B 0,C 180,E1 7210.202,E2 7210.202} C_VEL
LIN {X 0,Y 617.782,Z 1123.051,A -85,B 0,C 180,E1 7214.621,E2 7214.621} C_VEL
LIN {X 0,Y 617.566,Z 1132.642,A -85,B 0,C 180,E1 7219.158,E2 7219.158} C_VEL
LIN {X 0,Y 617.195,Z 1136.509,A -85,B 0,C 180,E1 7223.06,E2 7223.06} C_VEL
LIN {X 0,Y 617.207,Z 1136.751,A -85,B 0,C 180,E1 7226.145,E2 7226.145} C_VEL
LIN {X 0,Y 617.432,Z 1133.703,A -85,B 0,C 180,E1 7229.973,E2 7229.973} C_VEL
LIN {X 0,Y 617.844,Z 1125.82,A -85,B 0,C 180,E1 7234.227,E2 7234.227} C_VEL
LIN {X 0,Y 618.349,Z 1112.717,A -85,B 0,C 180,E1 7238.567,E2 7238.567} C_VEL
LIN {X 0,Y 619.261,Z 1093.465,A -85,B 0,C 180,E1 7243.093,E2 7243.093} C_VEL
LIN {X 0,Y 621.122,Z 1069.49,A -85,B 0,C 180,E1 7247.357,E2 7247.357} C_VEL
LIN {X 0,Y 623.865,Z 1039.943,A -85,B 0,C 180,E1 7251.493,E2 7251.493} C_VEL
LIN {X 0,Y 627.637,Z 1005.252,A -85,B 0,C 180,E1 7255.36,E2 7255.36} C_VEL
LIN {X 0,Y 632.198,Z 966.284,A -85,B 0,C 180,E1 7258.823,E2 7258.823} C_VEL
LIN {X 0,Y 637.06,Z 924.012,A -85,B 0,C 180,E1 7261.791,E2 7261.791} C_VEL
LIN {X 0,Y 641.709,Z 879.166,A -85,B 0,C 180,E1 7264.234,E2 7264.234} C_VEL
LIN {X 0,Y 642.19,Z 867.568,A -85,B 0,C 180,E1 7264.802,E2 7264.802} C_VEL
LIN {X 0,Y 627.001,Z 831.014,A -85,B 0,C 180,E1 7267.699,E2 7267.699} C_VEL
LIN {X 0,Y 616.889,Z 809.06,A -85,B 0,C 180,E1 7269.483,E2 7269.483} C_VEL
LIN {X 0,Y 617.056,Z 809.06,A -85,B 0,C 180,E1 7275.831,E2 7275.831} C_VEL
LIN {X 0,Y 617.336,Z 809.06,A -85,B 0,C 180,E1 7280.14,E2 7280.14} C_VEL
LIN {X 0,Y 617.462,Z 809.06,A -85,B 0,C 180,E1 7285.796,E2 7285.796} C_VEL
LIN {X 0,Y 617.588,Z 809.06,A -85,B 0,C 180,E1 7291.408,E2 7291.408} C_VEL
LIN {X 0,Y 617.344,Z 809.06,A -85,B 0,C 180,E1 7297.035,E2 7297.035} C_VEL
LIN {X 0,Y 617.265,Z 809.06,A -85,B 0,C 180,E1 7301.723,E2 7301.723} C_VEL
LIN {X 0,Y 617.212,Z 809.06,A -85,B 0,C 180,E1 7307.303,E2 7307.303} C_VEL
LIN {X 0,Y 617.019,Z 809.06,A -85,B 0,C 180,E1 7313.075,E2 7313.075} C_VEL
LIN {X 0,Y 616.929,Z 809.06,A -85,B 0,C 180,E1 7318.151,E2 7318.151} C_VEL
LIN {X 0,Y 616.893,Z 809.06,A -85,B 0,C 180,E1 7323.616,E2 7323.616} C_VEL
LIN {X 0,Y 616.759,Z 809.06,A -85,B 0,C 180,E1 7328.376,E2 7328.376} C_VEL
LIN {X 0,Y 616.864,Z 809.06,A -85,B 0,C 180,E1 7333.312,E2 7333.312} C_VEL
LIN {X 0,Y 616.793,Z 809.06,A -85,B 0,C 180,E1 7338.592,E2 7338.592} C_VEL
LIN {X 0,Y 616.786,Z 809.06,A -85,B 0,C 180,E1 7343.989,E2 7343.989} C_VEL
LIN {X 0,Y 616.852,Z 809.06,A -85,B 0,C 180,E1 7349.043,E2 7349.043} C_VEL
LIN {X 0,Y 617.085,Z 809.06,A -85,B 0,C 180,E1 7353.849,E2 7353.849} C_VEL
LIN {X 0,Y 617.148,Z 809.06,A -85,B 0,C 180,E1 7358.513,E2 7358.513} C_VEL
LIN {X 0,Y 617.202,Z 809.06,A -85,B 0,C 180,E1 7362.916,E2 7362.916} C_VEL
LIN {X 0,Y 617.28,Z 809.06,A -85,B 0,C 180,E1 7368.708,E2 7368.708} C_VEL
LIN {X 0,Y 617.41,Z 809.06,A -85,B 0,C 180,E1 7373.132,E2 7373.132} C_VEL
LIN {X 0,Y 617.511,Z 809.06,A -85,B 0,C 180,E1 7378.598,E2 7378.598} C_VEL
LIN {X 0,Y 617.493,Z 809.06,A -85,B 0,C 180,E1 7382.806,E2 7382.806} C_VEL
LIN {X 0,Y 617.38,Z 809.06,A -85,B 0,C 180,E1 7387.029,E2 7387.029} C_VEL
LIN {X 0,Y 617.242,Z 809.06,A -85,B 0,C 180,E1 7392.728,E2 7392.728} C_VEL
LIN {X 0,Y 617.176,Z 809.06,A -85,B 0,C 180,E1 7398.559,E2 7398.559} C_VEL
LIN {X 0,Y 617.021,Z 809.06,A -85,B 0,C 180,E1 7403.068,E2 7403.068} C_VEL
LIN {X 0,Y 616.893,Z 809.06,A -85,B 0,C 180,E1 7408.128,E2 7408.128} C_VEL
LIN {X 0,Y 616.886,Z 809.06,A -85,B 0,C 180,E1 7413.6,E2 7413.6} C_VEL
LIN {X 0,Y 616.778,Z 809.06,A -85,B 0,C 180,E1 7418.366,E2 7418.366} C_VEL
LIN {X 0,Y 616.923,Z 809.067,A -85,B 0,C 180,E1 7422.652,E2 7422.652} C_VEL
LIN {X 0,Y 619.358,Z 814.744,A -85,B 0,C 180,E1 7422.965,E2 7422.965} C_VEL
LIN {X 0,Y 633.28,Z 837.737,A -85,B 0,C 180,E1 7424.503,E2 7424.503} C_VEL
LIN {X 0,Y 638.519,Z 852.873,A -85,B 0,C 180,E1 7425.145,E2 7425.145} C_VEL
LIN {X 0,Y 643.438,Z 868.143,A -85,B 0,C 180,E1 7425.789,E2 7425.789} C_VEL
LIN {X 0,Y 645.271,Z 871.572,A -85,B 0,C 180,E1 7425.999,E2 7425.999} C_VEL
LIN {X 0,Y 643.485,Z 931.644,A -85,B 0,C 180,E1 7426.968,E2 7426.968} C_VEL
LIN {X 0,Y 640.176,Z 976.528,A -85,B 0,C 180,E1 7428.161,E2 7428.161} C_VEL
LIN {X 0,Y 636.127,Z 1022.317,A -85,B 0,C 180,E1 7429.95,E2 7429.95} C_VEL
LIN {X 0,Y 631.456,Z 1066.028,A -85,B 0,C 180,E1 7432.229,E2 7432.229} C_VEL
LIN {X 0,Y 626.287,Z 1108.57,A -85,B 0,C 180,E1 7435.115,E2 7435.115} C_VEL
LIN {X 0,Y 621.501,Z 1147.413,A -85,B 0,C 180,E1 7438.436,E2 7438.436} C_VEL
LIN {X 0,Y 617.096,Z 1184.182,A -85,B 0,C 180,E1 7442.406,E2 7442.406} C_VEL
LIN {X 0,Y 613.916,Z 1214.046,A -85,B 0,C 180,E1 7446.458,E2 7446.458} C_VEL
LIN {X 0,Y 611.68,Z 1239.805,A -85,B 0,C 180,E1 7450.888,E2 7450.888} C_VEL
LIN {X 0,Y 610.556,Z 1259.126,A -85,B 0,C 180,E1 7455.241,E2 7455.241} C_VEL
LIN {X 0,Y 609.988,Z 1272.346,A -85,B 0,C 180,E1 7459.287,E2 7459.287} C_VEL
LIN {X 0,Y 609.845,Z 1281.765,A -85,B 0,C 180,E1 7463.592,E2 7463.592} C_VEL
LIN {X 0,Y 609.729,Z 1285.872,A -85,B 0,C 180,E1 7467.153,E2 7467.153} C_VEL
LIN {X 0,Y 609.865,Z 1286.669,A -85,B 0,C 180,E1 7471.414,E2 7471.414} C_VEL
LIN {X 0,Y 609.717,Z 1282.919,A -85,B 0,C 180,E1 7475.683,E2 7475.683} C_VEL
LIN {X 0,Y 609.895,Z 1274.303,A -85,B 0,C 180,E1 7479.981,E2 7479.981} C_VEL
LIN {X 0,Y 610.562,Z 1260.736,A -85,B 0,C 180,E1 7484.323,E2 7484.323} C_VEL
LIN {X 0,Y 611.719,Z 1241.758,A -85,B 0,C 180,E1 7488.725,E2 7488.725} C_VEL
LIN {X 0,Y 613.815,Z 1216.29,A -85,B 0,C 180,E1 7493.19,E2 7493.19} C_VEL
LIN {X 0,Y 616.943,Z 1186.458,A -85,B 0,C 180,E1 7497.319,E2 7497.319} C_VEL
LIN {X 0,Y 621.1,Z 1150.724,A -85,B 0,C 180,E1 7501.235,E2 7501.235} C_VEL
LIN {X 0,Y 625.728,Z 1113.329,A -85,B 0,C 180,E1 7504.523,E2 7504.523} C_VEL
LIN {X 0,Y 630.873,Z 1070.253,A -85,B 0,C 180,E1 7507.513,E2 7507.513} C_VEL
LIN {X 0,Y 635.751,Z 1025.483,A -85,B 0,C 180,E1 7509.914,E2 7509.914} C_VEL
LIN {X 0,Y 640.177,Z 975.987,A -85,B 0,C 180,E1 7511.861,E2 7511.861} C_VEL
LIN {X 0,Y 643.369,Z 929.206,A -85,B 0,C 180,E1 7513.098,E2 7513.098} C_VEL
LIN {X 0,Y 644.975,Z 871.063,A -85,B 0,C 180,E1 7514.034,E2 7514.034} C_VEL
LIN {X 0,Y 631.153,Z 848.151,A -85,B 0,C 180,E1 7515.372,E2 7515.372} C_VEL
LIN {X 0,Y 616.832,Z 825.67,A -85,B 0,C 180,E1 7516.634,E2 7516.634} C_VEL
LIN {X 0,Y 608.972,Z 809.06,A -85,B 0,C 180,E1 7517.458,E2 7517.458} C_VEL
LIN {X 0,Y 608.841,Z 809.06,A -85,B 0,C 180,E1 7522.569,E2 7522.569} C_VEL
LIN {X 0,Y 608.866,Z 809.06,A -85,B 0,C 180,E1 7528.59,E2 7528.59} C_VEL
LIN {X 0,Y 608.916,Z 809.06,A -85,B 0,C 180,E1 7533.47,E2 7533.47} C_VEL
LIN {X 0,Y 608.935,Z 809.06,A -85,B 0,C 180,E1 7538.148,E2 7538.148} C_VEL
LIN {X 0,Y 609.024,Z 809.221,A -85,B 0,C 180,E1 7539.927,E2 7539.927} C_VEL
LIN {X 0,Y 623.883,Z 841.194,A -85,B 0,C 180,E1 7542.385,E2 7542.385} C_VEL
LIN {X 0,Y 636.124,Z 872.769,A -85,B 0,C 180,E1 7544.918,E2 7544.918} C_VEL
LIN {X 0,Y 631.129,Z 917.919,A -85,B 0,C 180,E1 7547.293,E2 7547.293} C_VEL
LIN {X 0,Y 626.002,Z 960.212,A -85,B 0,C 180,E1 7550.184,E2 7550.184} C_VEL
LIN {X 0,Y 621.34,Z 998.932,A -85,B 0,C 180,E1 7553.542,E2 7553.542} C_VEL
LIN {X 0,Y 617.187,Z 1034.233,A -85,B 0,C 180,E1 7557.368,E2 7557.368} C_VEL
LIN {X 0,Y 613.926,Z 1065.179,A -85,B 0,C 180,E1 7561.586,E2 7561.586} C_VEL
LIN {X 0,Y 611.803,Z 1088.93,A -85,B 0,C 180,E1 7565.669,E2 7565.669} C_VEL
LIN {X 0,Y 610.659,Z 1108.312,A -85,B 0,C 180,E1 7569.974,E2 7569.974} C_VEL
LIN {X 0,Y 609.902,Z 1122.671,A -85,B 0,C 180,E1 7574.343,E2 7574.343} C_VEL
LIN {X 0,Y 609.659,Z 1132.193,A -85,B 0,C 180,E1 7578.795,E2 7578.795} C_VEL
LIN {X 0,Y 609.261,Z 1136.678,A -85,B 0,C 180,E1 7583.43,E2 7583.43} C_VEL
LIN {X 0,Y 609.343,Z 1135.702,A -85,B 0,C 180,E1 7588.108,E2 7588.108} C_VEL
LIN {X 0,Y 609.739,Z 1129.617,A -85,B 0,C 180,E1 7592.597,E2 7592.597} C_VEL
LIN {X 0,Y 610.133,Z 1118.406,A -85,B 0,C 180,E1 7597.039,E2 7597.039} C_VEL
LIN {X 0,Y 611.013,Z 1101.373,A -85,B 0,C 180,E1 7601.617,E2 7601.617} C_VEL
LIN {X 0,Y 612.795,Z 1078.319,A -85,B 0,C 180,E1 7606.176,E2 7606.176} C_VEL
LIN {X 0,Y 615.495,Z 1050.012,A -85,B 0,C 180,E1 7610.513,E2 7610.513} C_VEL
LIN {X 0,Y 619.046,Z 1017.519,A -85,B 0,C 180,E1 7614.46,E2 7614.46} C_VEL
LIN {X 0,Y 623.513,Z 981.051,A -85,B 0,C 180,E1 7618.012,E2 7618.012} C_VEL
LIN {X 0,Y 628.522,Z 940.401,A -85,B 0,C 180,E1 7621.162,E2 7621.162} C_VEL
LIN {X 0,Y 633.572,Z 895.687,A -85,B 0,C 180,E1 7623.879,E2 7623.879} C_VEL
LIN {X 0,Y 635.979,Z 871.5,A -85,B 0,C 180,E1 7625.062,E2 7625.062} C_VEL
LIN {X 0,Y 620.821,Z 834.47,A -85,B 0,C 180,E1 7628.079,E2 7628.079} C_VEL
LIN {X 0,Y 608.967,Z 809.06,A -85,B 0,C 180,E1 7630.156,E2 7630.156} C_VEL
LIN {X 0,Y 609.12,Z 809.06,A -85,B 0,C 180,E1 7635.643,E2 7635.643} C_VEL
LIN {X 0,Y 609.413,Z 809.06,A -85,B 0,C 180,E1 7640.011,E2 7640.011} C_VEL
LIN {X 0,Y 609.553,Z 809.06,A -85,B 0,C 180,E1 7645.741,E2 7645.741} C_VEL
LIN {X 0,Y 609.682,Z 809.06,A -85,B 0,C 180,E1 7651.426,E2 7651.426} C_VEL
LIN {X 0,Y 609.436,Z 809.06,A -85,B 0,C 180,E1 7657.127,E2 7657.127} C_VEL
LIN {X 0,Y 609.383,Z 809.06,A -85,B 0,C 180,E1 7661.448,E2 7661.448} C_VEL
LIN {X 0,Y 609.317,Z 809.06,A -85,B 0,C 180,E1 7667.319,E2 7667.319} C_VEL
LIN {X 0,Y 609.147,Z 809.06,A -85,B 0,C 180,E1 7671.851,E2 7671.851} C_VEL
LIN {X 0,Y 609.028,Z 809.06,A -85,B 0,C 180,E1 7676.729,E2 7676.729} C_VEL
LIN {X 0,Y 608.995,Z 809.06,A -85,B 0,C 180,E1 7682.481,E2 7682.481} C_VEL
LIN {X 0,Y 608.89,Z 809.06,A -85,B 0,C 180,E1 7688.353,E2 7688.353} C_VEL
LIN {X 0,Y 608.928,Z 809.06,A -85,B 0,C 180,E1 7694.021,E2 7694.021} C_VEL
LIN {X 0,Y 608.856,Z 809.06,A -85,B 0,C 180,E1 7699.817,E2 7699.817} C_VEL
LIN {X 0,Y 608.822,Z 809.06,A -85,B 0,C 180,E1 7705.193,E2 7705.193} C_VEL
LIN {X 0,Y 609.022,Z 809.06,A -85,B 0,C 180,E1 7710.283,E2 7710.283} C_VEL
LIN {X 0,Y 609.163,Z 809.06,A -85,B 0,C 180,E1 7715.06,E2 7715.06} C_VEL
LIN {X 0,Y 609.222,Z 809.06,A -85,B 0,C 180,E1 7720.494,E2 7720.494} C_VEL
LIN {X 0,Y 609.258,Z 809.06,A -85,B 0,C 180,E1 7725.641,E2 7725.641} C_VEL
LIN {X 0,Y 609.517,Z 809.06,A -85,B 0,C 180,E1 7731.447,E2 7731.447} C_VEL
LIN {X 0,Y 609.673,Z 809.06,A -85,B 0,C 180,E1 7737.159,E2 7737.159} C_VEL
LIN {X 0,Y 609.827,Z 809.06,A -85,B 0,C 180,E1 7741.42,E2 7741.42} C_VEL
LIN {X 0,Y 609.472,Z 809.06,A -85,B 0,C 180,E1 7747.339,E2 7747.339} C_VEL
LIN {X 0,Y 609.321,Z 809.06,A -85,B 0,C 180,E1 7752.896,E2 7752.896} C_VEL
LIN {X 0,Y 609.294,Z 809.06,A -85,B 0,C 180,E1 7757.313,E2 7757.313} C_VEL
LIN {X 0,Y 609.151,Z 809.06,A -85,B 0,C 180,E1 7761.844,E2 7761.844} C_VEL
LIN {X 0,Y 608.984,Z 809.06,A -85,B 0,C 180,E1 7766.702,E2 7766.702} C_VEL
LIN {X 0,Y 608.974,Z 809.06,A -85,B 0,C 180,E1 7772.463,E2 7772.463} C_VEL
LIN {X 0,Y 608.909,Z 809.06,A -85,B 0,C 180,E1 7778.344,E2 7778.344} C_VEL
LIN {X 0,Y 608.967,Z 809.064,A -85,B 0,C 180,E1 7781.915,E2 7781.915} C_VEL
LIN {X 0,Y 611.26,Z 814.62,A -85,B 0,C 180,E1 7782.225,E2 7782.225} C_VEL
LIN {X 0,Y 643.438,Z 868.143,A -85,B 0,C 180,E1 7785.789,E2 7785.789} C_VEL
LIN {X 0,Y 643.798,Z 874.814,A -85,B 0,C 180,E1 7785.922,E2 7785.922} C_VEL
LIN {X 0,Y 639.202,Z 891.459,A -85,B 0,C 180,E1 7785.778,E2 7785.778} C_VEL
LIN {X 0,Y 636.901,Z 942.029,A -85,B 0,C 180,E1 7786.715,E2 7786.715} C_VEL
LIN {X 0,Y 633.42,Z 986.184,A -85,B 0,C 180,E1 7788.01,E2 7788.01} C_VEL
LIN {X 0,Y 628.973,Z 1031.654,A -85,B 0,C 180,E1 7789.912,E2 7789.912} C_VEL
LIN {X 0,Y 623.752,Z 1075.72,A -85,B 0,C 180,E1 7792.375,E2 7792.375} C_VEL
LIN {X 0,Y 618.586,Z 1116.658,A -85,B 0,C 180,E1 7795.313,E2 7795.313} C_VEL
LIN {X 0,Y 613.252,Z 1156.76,A -85,B 0,C 180,E1 7798.971,E2 7798.971} C_VEL
LIN {X 0,Y 609.027,Z 1190.727,A -85,B 0,C 180,E1 7802.872,E2 7802.872} C_VEL
LIN {X 0,Y 605.703,Z 1221.775,A -85,B 0,C 180,E1 7807.371,E2 7807.371} C_VEL
LIN {X 0,Y 603.628,Z 1246.458,A -85,B 0,C 180,E1 7812.03,E2 7812.03} C_VEL
LIN {X 0,Y 602.476,Z 1264.659,A -85,B 0,C 180,E1 7816.579,E2 7816.579} C_VEL
LIN {X 0,Y 601.876,Z 1277.679,A -85,B 0,C 180,E1 7821.33,E2 7821.33} C_VEL
LIN {X 0,Y 601.776,Z 1284.672,A -85,B 0,C 180,E1 7825.674,E2 7825.674} C_VEL
LIN {X 0,Y 601.837,Z 1287,A -85,B 0,C 180,E1 7829.994,E2 7829.994} C_VEL
LIN {X 0,Y 601.787,Z 1284.685,A -85,B 0,C 180,E1 7834.314,E2 7834.314} C_VEL
LIN {X 0,Y 601.83,Z 1277.705,A -85,B 0,C 180,E1 7838.658,E2 7838.658} C_VEL
LIN {X 0,Y 602.401,Z 1265.856,A -85,B 0,C 180,E1 7843.041,E2 7843.041} C_VEL
LIN {X 0,Y 603.419,Z 1248.736,A -85,B 0,C 180,E1 7847.481,E2 7847.481} C_VEL
LIN {X 0,Y 605.321,Z 1225.541,A -85,B 0,C 180,E1 7851.983,E2 7851.983} C_VEL
LIN {X 0,Y 608.273,Z 1198.097,A -85,B 0,C 180,E1 7856.157,E2 7856.157} C_VEL
LIN {X 0,Y 612.491,Z 1162.904,A -85,B 0,C 180,E1 7860.387,E2 7860.387} C_VEL
LIN {X 0,Y 617.252,Z 1125.816,A -85,B 0,C 180,E1 7863.927,E2 7863.927} C_VEL
LIN {X 0,Y 622.699,Z 1083.785,A -85,B 0,C 180,E1 7867.112,E2 7867.112} C_VEL
LIN {X 0,Y 628.008,Z 1039.592,A -85,B 0,C 180,E1 7869.692,E2 7869.692} C_VEL
LIN {X 0,Y 632.934,Z 992.285,A -85,B 0,C 180,E1 7871.773,E2 7871.773} C_VEL
LIN {X 0,Y 636.557,Z 946.587,A -85,B 0,C 180,E1 7873.179,E2 7873.179} C_VEL
LIN {X 0,Y 639.116,Z 897.97,A -85,B 0,C 180,E1 7874.116,E2 7874.116} C_VEL
LIN {X 0,Y 638.963,Z 873.893,A -85,B 0,C 180,E1 7874.51,E2 7874.51} C_VEL
LIN {X 0,Y 611.404,Z 830.343,A -85,B 0,C 180,E1 7876.944,E2 7876.944} C_VEL
LIN {X 0,Y 601.098,Z 810.07,A -85,B 0,C 180,E1 7877.992,E2 7877.992} C_VEL
LIN {X 0,Y 601.003,Z 809.06,A -85,B 0,C 180,E1 7878.106,E2 7878.106} C_VEL
LIN {X 0,Y 600.937,Z 809.06,A -85,B 0,C 180,E1 7883.565,E2 7883.565} C_VEL
LIN {X 0,Y 600.949,Z 809.06,A -85,B 0,C 180,E1 7888.738,E2 7888.738} C_VEL
LIN {X 0,Y 600.991,Z 809.06,A -85,B 0,C 180,E1 7893.092,E2 7893.092} C_VEL
LIN {X 0,Y 601.006,Z 809.06,A -85,B 0,C 180,E1 7898.923,E2 7898.923} C_VEL
LIN {X 0,Y 601.052,Z 809.631,A -85,B 0,C 180,E1 7899.276,E2 7899.276} C_VEL
LIN {X 0,Y 617.09,Z 843.478,A -85,B 0,C 180,E1 7901.93,E2 7901.93} C_VEL
LIN {X 0,Y 629.676,Z 875.176,A -85,B 0,C 180,E1 7904.557,E2 7904.557} C_VEL
LIN {X 0,Y 624.393,Z 920.185,A -85,B 0,C 180,E1 7906.976,E2 7906.976} C_VEL
LIN {X 0,Y 619.001,Z 962.063,A -85,B 0,C 180,E1 7909.895,E2 7909.895} C_VEL
LIN {X 0,Y 614.095,Z 1000.451,A -85,B 0,C 180,E1 7913.288,E2 7913.288} C_VEL
LIN {X 0,Y 609.721,Z 1035.478,A -85,B 0,C 180,E1 7917.159,E2 7917.159} C_VEL
LIN {X 0,Y 606.272,Z 1066.148,A -85,B 0,C 180,E1 7921.428,E2 7921.428} C_VEL
LIN {X 0,Y 603.909,Z 1090.599,A -85,B 0,C 180,E1 7925.743,E2 7925.743} C_VEL
LIN {X 0,Y 602.745,Z 1109.526,A -85,B 0,C 180,E1 7930.106,E2 7930.106} C_VEL
LIN {X 0,Y 601.999,Z 1123.557,A -85,B 0,C 180,E1 7934.536,E2 7934.536} C_VEL
LIN {X 0,Y 601.736,Z 1132.705,A -85,B 0,C 180,E1 7939.052,E2 7939.052} C_VEL
LIN {X 0,Y 601.351,Z 1136.749,A -85,B 0,C 180,E1 7943.704,E2 7943.704} C_VEL
LIN {X 0,Y 601.446,Z 1135.422,A -85,B 0,C 180,E1 7948.511,E2 7948.511} C_VEL
LIN {X 0,Y 601.883,Z 1128.964,A -85,B 0,C 180,E1 7953.02,E2 7953.02} C_VEL
LIN {X 0,Y 602.404,Z 1117.153,A -85,B 0,C 180,E1 7957.596,E2 7957.596} C_VEL
LIN {X 0,Y 603.402,Z 1099.815,A -85,B 0,C 180,E1 7962.197,E2 7962.197} C_VEL
LIN {X 0,Y 605.247,Z 1076.659,A -85,B 0,C 180,E1 7966.744,E2 7966.744} C_VEL
LIN {X 0,Y 608.191,Z 1048.411,A -85,B 0,C 180,E1 7971.069,E2 7971.069} C_VEL
LIN {X 0,Y 612.003,Z 1015.883,A -85,B 0,C 180,E1 7975.025,E2 7975.025} C_VEL
LIN {X 0,Y 616.979,Z 978.146,A -85,B 0,C 180,E1 7978.688,E2 7978.688} C_VEL
LIN {X 0,Y 622.506,Z 936.079,A -85,B 0,C 180,E1 7981.91,E2 7981.91} C_VEL
LIN {X 0,Y 627.834,Z 891.185,A -85,B 0,C 180,E1 7984.573,E2 7984.573} C_VEL
LIN {X 0,Y 629.285,Z 874.018,A -85,B 0,C 180,E1 7985.442,E2 7985.442} C_VEL
LIN {X 0,Y 614.409,Z 837.499,A -85,B 0,C 180,E1 7988.496,E2 7988.496} C_VEL
LIN {X 0,Y 601.007,Z 809.06,A -85,B 0,C 180,E1 7990.929,E2 7990.929} C_VEL
LIN {X 0,Y 601.316,Z 809.06,A -85,B 0,C 180,E1 7996.935,E2 7996.935} C_VEL
LIN {X 0,Y 601.566,Z 809.06,A -85,B 0,C 180,E1 8001.338,E2 8001.338} C_VEL
LIN {X 0,Y 601.772,Z 809.06,A -85,B 0,C 180,E1 8007.127,E2 8007.127} C_VEL
LIN {X 0,Y 601.776,Z 809.06,A -85,B 0,C 180,E1 8011.445,E2 8011.445} C_VEL
LIN {X 0,Y 601.552,Z 809.06,A -85,B 0,C 180,E1 8017.221,E2 8017.221} C_VEL
LIN {X 0,Y 601.452,Z 809.06,A -85,B 0,C 180,E1 8023.074,E2 8023.074} C_VEL
LIN {X 0,Y 601.381,Z 809.06,A -85,B 0,C 180,E1 8027.555,E2 8027.555} C_VEL
LIN {X 0,Y 601.203,Z 809.06,A -85,B 0,C 180,E1 8032.155,E2 8032.155} C_VEL
LIN {X 0,Y 601.109,Z 809.06,A -85,B 0,C 180,E1 8036.909,E2 8036.909} C_VEL
LIN {X 0,Y 601.066,Z 809.06,A -85,B 0,C 180,E1 8041.872,E2 8041.872} C_VEL
LIN {X 0,Y 600.963,Z 809.06,A -85,B 0,C 180,E1 8047.125,E2 8047.125} C_VEL
LIN {X 0,Y 600.953,Z 809.06,A -85,B 0,C 180,E1 8053.185,E2 8053.185} C_VEL
LIN {X 0,Y 600.904,Z 809.06,A -85,B 0,C 180,E1 8059.174,E2 8059.174} C_VEL
LIN {X 0,Y 600.916,Z 809.06,A -85,B 0,C 180,E1 8064.668,E2 8064.668} C_VEL
LIN {X 0,Y 601.035,Z 809.06,A -85,B 0,C 180,E1 8069.816,E2 8069.816} C_VEL
LIN {X 0,Y 601.231,Z 809.06,A -85,B 0,C 180,E1 8074.806,E2 8074.806} C_VEL
LIN {X 0,Y 601.284,Z 809.06,A -85,B 0,C 180,E1 8079.402,E2 8079.402} C_VEL
LIN {X 0,Y 601.357,Z 809.06,A -85,B 0,C 180,E1 8083.956,E2 8083.956} C_VEL
LIN {X 0,Y 601.488,Z 809.06,A -85,B 0,C 180,E1 8089.873,E2 8089.873} C_VEL
LIN {X 0,Y 601.593,Z 809.06,A -85,B 0,C 180,E1 8094.235,E2 8094.235} C_VEL
LIN {X 0,Y 601.884,Z 809.06,A -85,B 0,C 180,E1 8100.001,E2 8100.001} C_VEL
LIN {X 0,Y 601.665,Z 809.06,A -85,B 0,C 180,E1 8105.766,E2 8105.766} C_VEL
LIN {X 0,Y 601.469,Z 809.06,A -85,B 0,C 180,E1 8111.594,E2 8111.594} C_VEL
LIN {X 0,Y 601.38,Z 809.06,A -85,B 0,C 180,E1 8117.549,E2 8117.549} C_VEL
LIN {X 0,Y 601.214,Z 809.06,A -85,B 0,C 180,E1 8122.148,E2 8122.148} C_VEL
LIN {X 0,Y 601.067,Z 809.06,A -85,B 0,C 180,E1 8126.904,E2 8126.904} C_VEL
LIN {X 0,Y 601.052,Z 809.06,A -85,B 0,C 180,E1 8131.866,E2 8131.866} C_VEL
LIN {X 0,Y 600.975,Z 809.06,A -85,B 0,C 180,E1 8137.116,E2 8137.116} C_VEL
LIN {X 0,Y 600.985,Z 809.06,A -85,B 0,C 180,E1 8141.121,E2 8141.121} C_VEL
LIN {X 0,Y 603.558,Z 814.872,A -85,B 0,C 180,E1 8141.499,E2 8141.499} C_VEL
LIN {X 0,Y 639.268,Z 874.413,A -85,B 0,C 180,E1 8145.523,E2 8145.523} C_VEL
LIN {X 0,Y 639.202,Z 891.459,A -85,B 0,C 180,E1 8145.778,E2 8145.778} C_VEL
LIN {X 0,Y 635.756,Z 908.669,A -85,B 0,C 180,E1 8145.79,E2 8145.79} C_VEL
LIN {X 0,Y 632.151,Z 925.779,A -85,B 0,C 180,E1 8145.88,E2 8145.88} C_VEL
LIN {X 0,Y 628.896,Z 970.424,A -85,B 0,C 180,E1 8146.988,E2 8146.988} C_VEL
LIN {X 0,Y 624.747,Z 1014.24,A -85,B 0,C 180,E1 8148.632,E2 8148.632} C_VEL
LIN {X 0,Y 619.429,Z 1059.304,A -85,B 0,C 180,E1 8150.91,E2 8150.91} C_VEL
LIN {X 0,Y 613.829,Z 1101.333,A -85,B 0,C 180,E1 8153.675,E2 8153.675} C_VEL
LIN {X 0,Y 608.143,Z 1142.444,A -85,B 0,C 180,E1 8157.145,E2 8157.145} C_VEL
LIN {X 0,Y 603.345,Z 1177.781,A -85,B 0,C 180,E1 8160.903,E2 8160.903} C_VEL
LIN {X 0,Y 599.209,Z 1210.696,A -85,B 0,C 180,E1 8165.3,E2 8165.3} C_VEL
LIN {X 0,Y 596.527,Z 1237.11,A -85,B 0,C 180,E1 8169.849,E2 8169.849} C_VEL
LIN {X 0,Y 595.05,Z 1256.188,A -85,B 0,C 180,E1 8174.072,E2 8174.072} C_VEL
LIN {X 0,Y 594.295,Z 1270.403,A -85,B 0,C 180,E1 8178.258,E2 8178.258} C_VEL
LIN {X 0,Y 593.984,Z 1280.727,A -85,B 0,C 180,E1 8182.793,E2 8182.793} C_VEL
LIN {X 0,Y 593.934,Z 1285.871,A -85,B 0,C 180,E1 8187.077,E2 8187.077} C_VEL
LIN {X 0,Y 594.084,Z 1286.669,A -85,B 0,C 180,E1 8191.452,E2 8191.452} C_VEL
LIN {X 0,Y 593.932,Z 1282.919,A -85,B 0,C 180,E1 8195.835,E2 8195.835} C_VEL
LIN {X 0,Y 594.165,Z 1274.302,A -85,B 0,C 180,E1 8200.248,E2 8200.248} C_VEL
LIN {X 0,Y 594.871,Z 1260.735,A -85,B 0,C 180,E1 8204.709,E2 8204.709} C_VEL
LIN {X 0,Y 596.188,Z 1241.76,A -85,B 0,C 180,E1 8209.231,E2 8209.231} C_VEL
LIN {X 0,Y 598.656,Z 1216.286,A -85,B 0,C 180,E1 8213.813,E2 8213.813} C_VEL
LIN {X 0,Y 602.217,Z 1186.356,A -85,B 0,C 180,E1 8218.058,E2 8218.058} C_VEL
LIN {X 0,Y 607.194,Z 1149.109,A -85,B 0,C 180,E1 8222.211,E2 8222.211} C_VEL
LIN {X 0,Y 612.366,Z 1112.212,A -85,B 0,C 180,E1 8225.485,E2 8225.485} C_VEL
LIN {X 0,Y 618.117,Z 1069.444,A -85,B 0,C 180,E1 8228.485,E2 8228.485} C_VEL
LIN {X 0,Y 623.464,Z 1025.476,A -85,B 0,C 180,E1 8230.865,E2 8230.865} C_VEL
LIN {X 0,Y 628.252,Z 977.132,A -85,B 0,C 180,E1 8232.794,E2 8232.794} C_VEL
LIN {X 0,Y 631.713,Z 930.538,A -85,B 0,C 180,E1 8234.044,E2 8234.044} C_VEL
LIN {X 0,Y 632.919,Z 877.464,A -85,B 0,C 180,E1 8234.867,E2 8234.867} C_VEL
LIN {X 0,Y 606.019,Z 835.034,A -85,B 0,C 180,E1 8237.261,E2 8237.261} C_VEL
LIN {X 0,Y 593.136,Z 810.163,A -85,B 0,C 180,E1 8238.609,E2 8238.609} C_VEL
LIN {X 0,Y 593.032,Z 809.06,A -85,B 0,C 180,E1 8238.688,E2 8238.688} C_VEL
LIN {X 0,Y 593.007,Z 809.06,A -85,B 0,C 180,E1 8244.616,E2 8244.616} C_VEL
LIN {X 0,Y 593.031,Z 809.06,A -85,B 0,C 180,E1 8250.022,E2 8250.022} C_VEL
LIN {X 0,Y 593.073,Z 809.06,A -85,B 0,C 180,E1 8254.334,E2 8254.334} C_VEL
LIN {X 0,Y 593.128,Z 809.552,A -85,B 0,C 180,E1 8258.585,E2 8258.585} C_VEL
LIN {X 0,Y 610.556,Z 846.343,A -85,B 0,C 180,E1 8261.519,E2 8261.519} C_VEL
LIN {X 0,Y 623.127,Z 878.82,A -85,B 0,C 180,E1 8264.252,E2 8264.252} C_VEL
LIN {X 0,Y 617.692,Z 922.44,A -85,B 0,C 180,E1 8266.652,E2 8266.652} C_VEL
LIN {X 0,Y 612.025,Z 963.909,A -85,B 0,C 180,E1 8269.599,E2 8269.599} C_VEL
LIN {X 0,Y 606.614,Z 1003.725,A -85,B 0,C 180,E1 8273.205,E2 8273.205} C_VEL
LIN {X 0,Y 602.057,Z 1038.074,A -85,B 0,C 180,E1 8277.122,E2 8277.122} C_VEL
LIN {X 0,Y 598.459,Z 1068.23,A -85,B 0,C 180,E1 8281.446,E2 8281.446} C_VEL
LIN {X 0,Y 596.045,Z 1092.202,A -85,B 0,C 180,E1 8285.819,E2 8285.819} C_VEL
LIN {X 0,Y 594.837,Z 1110.74,A -85,B 0,C 180,E1 8290.242,E2 8290.242} C_VEL
LIN {X 0,Y 594.087,Z 1124.408,A -85,B 0,C 180,E1 8294.734,E2 8294.734} C_VEL
LIN {X 0,Y 593.864,Z 1132.063,A -85,B 0,C 180,E1 8298.544,E2 8298.544} C_VEL
LIN {X 0,Y 593.464,Z 1136.209,A -85,B 0,C 180,E1 8302.451,E2 8302.451} C_VEL
LIN {X 0,Y 593.458,Z 1136.307,A -85,B 0,C 180,E1 8307.276,E2 8307.276} C_VEL
LIN {X 0,Y 593.892,Z 1132.327,A -85,B 0,C 180,E1 8311.192,E2 8311.192} C_VEL
LIN {X 0,Y 594.214,Z 1122.826,A -85,B 0,C 180,E1 8315.792,E2 8315.792} C_VEL
LIN {X 0,Y 594.846,Z 1109.898,A -85,B 0,C 180,E1 8319.9,E2 8319.9} C_VEL
LIN {X 0,Y 596.117,Z 1091.87,A -85,B 0,C 180,E1 8324.16,E2 8324.16} C_VEL
LIN {X 0,Y 598.498,Z 1067.735,A -85,B 0,C 180,E1 8328.541,E2 8328.541} C_VEL
LIN {X 0,Y 601.928,Z 1038.682,A -85,B 0,C 180,E1 8332.709,E2 8332.709} C_VEL
LIN {X 0,Y 606.465,Z 1004.31,A -85,B 0,C 180,E1 8336.645,E2 8336.645} C_VEL
LIN {X 0,Y 611.91,Z 965.727,A -85,B 0,C 180,E1 8340.159,E2 8340.159} C_VEL
LIN {X 0,Y 617.668,Z 923.491,A -85,B 0,C 180,E1 8343.19,E2 8343.19} C_VEL
LIN {X 0,Y 622.959,Z 880.497,A -85,B 0,C 180,E1 8345.582,E2 8345.582} C_VEL
LIN {X 0,Y 621.245,Z 872.633,A -85,B 0,C 180,E1 8346.155,E2 8346.155} C_VEL
LIN {X 0,Y 605.576,Z 835.33,A -85,B 0,C 180,E1 8349.369,E2 8349.369} C_VEL
LIN {X 0,Y 593.134,Z 810.07,A -85,B 0,C 180,E1 8351.582,E2 8351.582} C_VEL
LIN {X 0,Y 593.058,Z 809.06,A -85,B 0,C 180,E1 8351.82,E2 8351.82} C_VEL
LIN {X 0,Y 593.38,Z 809.06,A -85,B 0,C 180,E1 8356.757,E2 8356.757} C_VEL
LIN {X 0,Y 593.666,Z 809.06,A -85,B 0,C 180,E1 8361.222,E2 8361.222} C_VEL
LIN {X 0,Y 593.864,Z 809.06,A -85,B 0,C 180,E1 8367.089,E2 8367.089} C_VEL
LIN {X 0,Y 593.87,Z 809.06,A -85,B 0,C 180,E1 8371.464,E2 8371.464} C_VEL
LIN {X 0,Y 593.661,Z 809.06,A -85,B 0,C 180,E1 8377.318,E2 8377.318} C_VEL
LIN {X 0,Y 593.554,Z 809.06,A -85,B 0,C 180,E1 8381.757,E2 8381.757} C_VEL
LIN {X 0,Y 593.486,Z 809.06,A -85,B 0,C 180,E1 8386.27,E2 8386.27} C_VEL
LIN {X 0,Y 593.357,Z 809.06,A -85,B 0,C 180,E1 8390.893,E2 8390.893} C_VEL
LIN {X 0,Y 593.223,Z 809.06,A -85,B 0,C 180,E1 8396.942,E2 8396.942} C_VEL
LIN {X 0,Y 593.08,Z 809.06,A -85,B 0,C 180,E1 8402.783,E2 8402.783} C_VEL
LIN {X 0,Y 593.004,Z 809.06,A -85,B 0,C 180,E1 8407.826,E2 8407.826} C_VEL
LIN {X 0,Y 593.014,Z 809.06,A -85,B 0,C 180,E1 8413.479,E2 8413.479} C_VEL
LIN {X 0,Y 592.964,Z 809.06,A -85,B 0,C 180,E1 8418.508,E2 8418.508} C_VEL
LIN {X 0,Y 593.029,Z 809.06,A -85,B 0,C 180,E1 8424.634,E2 8424.634} C_VEL
LIN {X 0,Y 593.128,Z 809.06,A -85,B 0,C 180,E1 8430.03,E2 8430.03} C_VEL
LIN {X 0,Y 593.283,Z 809.06,A -85,B 0,C 180,E1 8434.345,E2 8434.345} C_VEL
LIN {X 0,Y 593.376,Z 809.06,A -85,B 0,C 180,E1 8439.115,E2 8439.115} C_VEL
LIN {X 0,Y 593.451,Z 809.06,A -85,B 0,C 180,E1 8443.736,E2 8443.736} C_VEL
LIN {X 0,Y 593.591,Z 809.06,A -85,B 0,C 180,E1 8449.736,E2 8449.736} C_VEL
LIN {X 0,Y 593.687,Z 809.06,A -85,B 0,C 180,E1 8454.158,E2 8454.158} C_VEL
LIN {X 0,Y 593.983,Z 809.06,A -85,B 0,C 180,E1 8460.001,E2 8460.001} C_VEL
LIN {X 0,Y 593.751,Z 809.06,A -85,B 0,C 180,E1 8465.843,E2 8465.843} C_VEL
LIN {X 0,Y 593.543,Z 809.06,A -85,B 0,C 180,E1 8471.751,E2 8471.751} C_VEL
LIN {X 0,Y 593.463,Z 809.06,A -85,B 0,C 180,E1 8476.265,E2 8476.265} C_VEL
LIN {X 0,Y 593.344,Z 809.06,A -85,B 0,C 180,E1 8480.887,E2 8480.887} C_VEL
LIN {X 0,Y 593.193,Z 809.06,A -85,B 0,C 180,E1 8486.917,E2 8486.917} C_VEL
LIN {X 0,Y 593.071,Z 809.06,A -85,B 0,C 180,E1 8492.766,E2 8492.766} C_VEL
LIN {X 0,Y 593.02,Z 809.06,A -85,B 0,C 180,E1 8497.815,E2 8497.815} C_VEL
LIN {X 0,Y 593.014,Z 809.06,A -85,B 0,C 180,E1 8500.342,E2 8500.342} C_VEL
LIN {X 0,Y 595.3,Z 814.602,A -85,B 0,C 180,E1 8500.679,E2 8500.679} C_VEL
LIN {X 0,Y 629.304,Z 870.801,A -85,B 0,C 180,E1 8504.673,E2 8504.673} C_VEL
LIN {X 0,Y 633.31,Z 877.59,A -85,B 0,C 180,E1 8505.098,E2 8505.098} C_VEL
LIN {X 0,Y 632.151,Z 925.779,A -85,B 0,C 180,E1 8505.88,E2 8505.88} C_VEL
LIN {X 0,Y 628.027,Z 942.795,A -85,B 0,C 180,E1 8506.005,E2 8506.005} C_VEL
LIN {X 0,Y 623.844,Z 957.505,A -85,B 0,C 180,E1 8506.145,E2 8506.145} C_VEL
LIN {X 0,Y 623.61,Z 959.607,A -85,B 0,C 180,E1 8506.199,E2 8506.199} C_VEL
LIN {X 0,Y 619.64,Z 1004.987,A -85,B 0,C 180,E1 8507.74,E2 8507.74} C_VEL
LIN {X 0,Y 614.242,Z 1050.399,A -85,B 0,C 180,E1 8509.916,E2 8509.916} C_VEL
LIN {X 0,Y 607.942,Z 1096.098,A -85,B 0,C 180,E1 8512.827,E2 8512.827} C_VEL
LIN {X 0,Y 602.156,Z 1135.992,A -85,B 0,C 180,E1 8516.113,E2 8516.113} C_VEL
LIN {X 0,Y 596.793,Z 1173.398,A -85,B 0,C 180,E1 8519.989,E2 8519.989} C_VEL
LIN {X 0,Y 592.416,Z 1206.105,A -85,B 0,C 180,E1 8524.297,E2 8524.297} C_VEL
LIN {X 0,Y 589.448,Z 1231.964,A -85,B 0,C 180,E1 8528.568,E2 8528.568} C_VEL
LIN {X 0,Y 587.481,Z 1253.452,A -85,B 0,C 180,E1 8533.174,E2 8533.174} C_VEL
LIN {X 0,Y 586.462,Z 1269.263,A -85,B 0,C 180,E1 8537.721,E2 8537.721} C_VEL
LIN {X 0,Y 586.088,Z 1279.21,A -85,B 0,C 180,E1 8541.842,E2 8541.842} C_VEL
LIN {X 0,Y 585.984,Z 1284.667,A -85,B 0,C 180,E1 8545.557,E2 8545.557} C_VEL
LIN {X 0,Y 586.048,Z 1287,A -85,B 0,C 180,E1 8549.994,E2 8549.994} C_VEL
LIN {X 0,Y 585.99,Z 1284.682,A -85,B 0,C 180,E1 8554.431,E2 8554.431} C_VEL
LIN {X 0,Y 586.05,Z 1279.234,A -85,B 0,C 180,E1 8558.146,E2 8558.146} C_VEL
LIN {X 0,Y 586.589,Z 1268.157,A -85,B 0,C 180,E1 8562.642,E2 8562.642} C_VEL
LIN {X 0,Y 587.601,Z 1251.96,A -85,B 0,C 180,E1 8567.195,E2 8567.195} C_VEL
LIN {X 0,Y 589.597,Z 1229.869,A -85,B 0,C 180,E1 8571.809,E2 8571.809} C_VEL
LIN {X 0,Y 593.118,Z 1200.663,A -85,B 0,C 180,E1 8576.502,E2 8576.502} C_VEL
LIN {X 0,Y 597.487,Z 1168.276,A -85,B 0,C 180,E1 8580.586,E2 8580.586} C_VEL
LIN {X 0,Y 602.994,Z 1130.426,A -85,B 0,C 180,E1 8584.404,E2 8584.404} C_VEL
LIN {X 0,Y 608.975,Z 1088.555,A -85,B 0,C 180,E1 8587.708,E2 8587.708} C_VEL
LIN {X 0,Y 614.998,Z 1044.758,A -85,B 0,C 180,E1 8590.39,E2 8590.39} C_VEL
LIN {X 0,Y 620.479,Z 997.594,A -85,B 0,C 180,E1 8592.549,E2 8592.549} C_VEL
LIN {X 0,Y 623.734,Z 956.74,A -85,B 0,C 180,E1 8593.844,E2 8593.844} C_VEL
LIN {X 0,Y 626.251,Z 908.95,A -85,B 0,C 180,E1 8594.822,E2 8594.822} C_VEL
LIN {X 0,Y 626.243,Z 880.292,A -85,B 0,C 180,E1 8595.255,E2 8595.255} C_VEL
LIN {X 0,Y 600.969,Z 840.338,A -85,B 0,C 180,E1 8597.551,E2 8597.551} C_VEL
LIN {X 0,Y 585.244,Z 810.423,A -85,B 0,C 180,E1 8599.248,E2 8599.248} C_VEL
LIN {X 0,Y 585.111,Z 809.06,A -85,B 0,C 180,E1 8599.348,E2 8599.348} C_VEL
LIN {X 0,Y 585.077,Z 809.06,A -85,B 0,C 180,E1 8605.725,E2 8605.725} C_VEL
LIN {X 0,Y 585.126,Z 809.06,A -85,B 0,C 180,E1 8611.392,E2 8611.392} C_VEL
LIN {X 0,Y 585.149,Z 809.06,A -85,B 0,C 180,E1 8617.211,E2 8617.211} C_VEL
LIN {X 0,Y 585.21,Z 809.239,A -85,B 0,C 180,E1 8617.851,E2 8617.851} C_VEL
LIN {X 0,Y 592.132,Z 824.296,A -85,B 0,C 180,E1 8619.016,E2 8619.016} C_VEL
LIN {X 0,Y 609.253,Z 861.171,A -85,B 0,C 180,E1 8622.134,E2 8622.134} C_VEL
LIN {X 0,Y 616.569,Z 882.488,A -85,B 0,C 180,E1 8623.939,E2 8623.939} C_VEL
LIN {X 0,Y 610.641,Z 927.447,A -85,B 0,C 180,E1 8626.495,E2 8626.495} C_VEL
LIN {X 0,Y 604.49,Z 969.991,A -85,B 0,C 180,E1 8629.65,E2 8629.65} C_VEL
LIN {X 0,Y 598.857,Z 1008.582,A -85,B 0,C 180,E1 8633.298,E2 8633.298} C_VEL
LIN {X 0,Y 594.125,Z 1042.006,A -85,B 0,C 180,E1 8637.266,E2 8637.266} C_VEL
LIN {X 0,Y 590.542,Z 1071.515,A -85,B 0,C 180,E1 8641.671,E2 8641.671} C_VEL
LIN {X 0,Y 588.016,Z 1095.521,A -85,B 0,C 180,E1 8646.269,E2 8646.269} C_VEL
LIN {X 0,Y 586.842,Z 1113.241,A -85,B 0,C 180,E1 8650.748,E2 8650.748} C_VEL
LIN {X 0,Y 586.206,Z 1125.224,A -85,B 0,C 180,E1 8654.936,E2 8654.936} C_VEL
LIN {X 0,Y 585.941,Z 1132.586,A -85,B 0,C 180,E1 8658.804,E2 8658.804} C_VEL
LIN {X 0,Y 585.541,Z 1136.402,A -85,B 0,C 180,E1 8662.772,E2 8662.772} C_VEL
LIN {X 0,Y 585.498,Z 1136.801,A -85,B 0,C 180,E1 8666.021,E2 8666.021} C_VEL
LIN {X 0,Y 585.888,Z 1133.387,A -85,B 0,C 180,E1 8670.484,E2 8670.484} C_VEL
LIN {X 0,Y 586.287,Z 1126.249,A -85,B 0,C 180,E1 8674.54,E2 8674.54} C_VEL
LIN {X 0,Y 586.913,Z 1113.676,A -85,B 0,C 180,E1 8679.036,E2 8679.036} C_VEL
LIN {X 0,Y 588.214,Z 1094.266,A -85,B 0,C 180,E1 8683.913,E2 8683.913} C_VEL
LIN {X 0,Y 590.567,Z 1071.146,A -85,B 0,C 180,E1 8688.307,E2 8688.307} C_VEL
LIN {X 0,Y 594.317,Z 1041.101,A -85,B 0,C 180,E1 8692.766,E2 8692.766} C_VEL
LIN {X 0,Y 599.046,Z 1006.847,A -85,B 0,C 180,E1 8696.797,E2 8696.797} C_VEL
LIN {X 0,Y 604.73,Z 968.647,A -85,B 0,C 180,E1 8700.366,E2 8700.366} C_VEL
LIN {X 0,Y 610.536,Z 928.532,A -85,B 0,C 180,E1 8703.335,E2 8703.335} C_VEL
LIN {X 0,Y 616.052,Z 886.268,A -85,B 0,C 180,E1 8705.784,E2 8705.784} C_VEL
LIN {X 0,Y 616.24,Z 879.764,A -85,B 0,C 180,E1 8706.165,E2 8706.165} C_VEL
LIN {X 0,Y 601.342,Z 842.951,A -85,B 0,C 180,E1 8709.409,E2 8709.409} C_VEL
LIN {X 0,Y 585.226,Z 809.891,A -85,B 0,C 180,E1 8712.384,E2 8712.384} C_VEL
LIN {X 0,Y 585.229,Z 809.06,A -85,B 0,C 180,E1 8713.506,E2 8713.506} C_VEL
LIN {X 0,Y 585.617,Z 809.06,A -85,B 0,C 180,E1 8718.653,E2 8718.653} C_VEL
LIN {X 0,Y 585.816,Z 809.06,A -85,B 0,C 180,E1 8724.084,E2 8724.084} C_VEL
LIN {X 0,Y 585.861,Z 809.06,A -85,B 0,C 180,E1 8728.528,E2 8728.528} C_VEL
LIN {X 0,Y 585.797,Z 809.06,A -85,B 0,C 180,E1 8732.963,E2 8732.963} C_VEL
LIN {X 0,Y 585.75,Z 809.06,A -85,B 0,C 180,E1 8737.417,E2 8737.417} C_VEL
LIN {X 0,Y 585.632,Z 809.06,A -85,B 0,C 180,E1 8741.919,E2 8741.919} C_VEL
LIN {X 0,Y 585.535,Z 809.06,A -85,B 0,C 180,E1 8747.296,E2 8747.296} C_VEL
LIN {X 0,Y 585.338,Z 809.06,A -85,B 0,C 180,E1 8752.788,E2 8752.788} C_VEL
LIN {X 0,Y 585.222,Z 809.06,A -85,B 0,C 180,E1 8758.617,E2 8758.617} C_VEL
LIN {X 0,Y 585.158,Z 809.06,A -85,B 0,C 180,E1 8764.625,E2 8764.625} C_VEL
LIN {X 0,Y 585.08,Z 809.06,A -85,B 0,C 180,E1 8770.223,E2 8770.223} C_VEL
LIN {X 0,Y 585.099,Z 809.06,A -85,B 0,C 180,E1 8775.793,E2 8775.793} C_VEL
LIN {X 0,Y 585.012,Z 809.06,A -85,B 0,C 180,E1 8781.693,E2 8781.693} C_VEL
LIN {X 0,Y 585.098,Z 809.06,A -85,B 0,C 180,E1 8787.159,E2 8787.159} C_VEL
LIN {X 0,Y 585.296,Z 809.06,A -85,B 0,C 180,E1 8792.311,E2 8792.311} C_VEL
LIN {X 0,Y 585.382,Z 809.06,A -85,B 0,C 180,E1 8797.221,E2 8797.221} C_VEL
LIN {X 0,Y 585.528,Z 809.06,A -85,B 0,C 180,E1 8802.736,E2 8802.736} C_VEL
LIN {X 0,Y 585.612,Z 809.06,A -85,B 0,C 180,E1 8808.699,E2 8808.699} C_VEL
LIN {X 0,Y 585.813,Z 809.06,A -85,B 0,C 180,E1 8814.079,E2 8814.079} C_VEL
LIN {X 0,Y 586.096,Z 809.06,A -85,B 0,C 180,E1 8820.001,E2 8820.001} C_VEL
LIN {X 0,Y 585.867,Z 809.06,A -85,B 0,C 180,E1 8825.922,E2 8825.922} C_VEL
LIN {X 0,Y 585.632,Z 809.06,A -85,B 0,C 180,E1 8831.912,E2 8831.912} C_VEL
LIN {X 0,Y 585.532,Z 809.06,A -85,B 0,C 180,E1 8837.265,E2 8837.265} C_VEL
LIN {X 0,Y 585.334,Z 809.06,A -85,B 0,C 180,E1 8842.782,E2 8842.782} C_VEL
LIN {X 0,Y 585.187,Z 809.06,A -85,B 0,C 180,E1 8848.593,E2 8848.593} C_VEL
LIN {X 0,Y 585.164,Z 809.06,A -85,B 0,C 180,E1 8854.617,E2 8854.617} C_VEL
LIN {X 0,Y 585.118,Z 809.152,A -85,B 0,C 180,E1 8859.543,E2 8859.543} C_VEL
LIN {X 0,Y 587.463,Z 814.7,A -85,B 0,C 180,E1 8859.885,E2 8859.885} C_VEL
LIN {X 0,Y 617.64,Z 864.365,A -85,B 0,C 180,E1 8863.597,E2 8863.597} C_VEL
LIN {X 0,Y 627.425,Z 881.003,A -85,B 0,C 180,E1 8864.673,E2 8864.673} C_VEL
LIN {X 0,Y 625.648,Z 934.346,A -85,B 0,C 180,E1 8865.59,E2 8865.59} C_VEL
LIN {X 0,Y 623.61,Z 959.607,A -85,B 0,C 180,E1 8866.199,E2 8866.199} C_VEL
LIN {X 0,Y 614.924,Z 990.842,A -85,B 0,C 180,E1 8866.736,E2 8866.736} C_VEL
LIN {X 0,Y 614.609,Z 992.848,A -85,B 0,C 180,E1 8866.806,E2 8866.806} C_VEL
LIN {X 0,Y 609.741,Z 1037.659,A -85,B 0,C 180,E1 8868.748,E2 8868.748} C_VEL
LIN {X 0,Y 603.601,Z 1082.259,A -85,B 0,C 180,E1 8871.38,E2 8871.38} C_VEL
LIN {X 0,Y 597.547,Z 1122.042,A -85,B 0,C 180,E1 8874.429,E2 8874.429} C_VEL
LIN {X 0,Y 591.717,Z 1159.299,A -85,B 0,C 180,E1 8877.995,E2 8877.995} C_VEL
LIN {X 0,Y 586.544,Z 1193.744,A -85,B 0,C 180,E1 8882.174,E2 8882.174} C_VEL
LIN {X 0,Y 582.825,Z 1222.57,A -85,B 0,C 180,E1 8886.574,E2 8886.574} C_VEL
LIN {X 0,Y 580.267,Z 1246.945,A -85,B 0,C 180,E1 8891.391,E2 8891.391} C_VEL
LIN {X 0,Y 578.985,Z 1264.661,A -85,B 0,C 180,E1 8896.024,E2 8896.024} C_VEL
LIN {X 0,Y 578.251,Z 1277.67,A -85,B 0,C 180,E1 8900.973,E2 8900.973} C_VEL
LIN {X 0,Y 578.082,Z 1284.664,A -85,B 0,C 180,E1 8905.496,E2 8905.496} C_VEL
LIN {X 0,Y 578.148,Z 1287,A -85,B 0,C 180,E1 8909.994,E2 8909.994} C_VEL
LIN {X 0,Y 578.086,Z 1284.679,A -85,B 0,C 180,E1 8914.491,E2 8914.491} C_VEL
LIN {X 0,Y 578.211,Z 1277.696,A -85,B 0,C 180,E1 8919.015,E2 8919.015} C_VEL
LIN {X 0,Y 578.889,Z 1265.859,A -85,B 0,C 180,E1 8923.581,E2 8923.581} C_VEL
LIN {X 0,Y 580.211,Z 1248.731,A -85,B 0,C 180,E1 8928.204,E2 8928.204} C_VEL
LIN {X 0,Y 582.752,Z 1223.918,A -85,B 0,C 180,E1 8933.181,E2 8933.181} C_VEL
LIN {X 0,Y 586.388,Z 1195.181,A -85,B 0,C 180,E1 8937.628,E2 8937.628} C_VEL
LIN {X 0,Y 591.412,Z 1161.257,A -85,B 0,C 180,E1 8941.794,E2 8941.794} C_VEL
LIN {X 0,Y 597.226,Z 1123.608,A -85,B 0,C 180,E1 8945.442,E2 8945.442} C_VEL
LIN {X 0,Y 603.525,Z 1082.439,A -85,B 0,C 180,E1 8948.613,E2 8948.613} C_VEL
LIN {X 0,Y 609.817,Z 1036.483,A -85,B 0,C 180,E1 8951.319,E2 8951.319} C_VEL
LIN {X 0,Y 613.917,Z 997.739,A -85,B 0,C 180,E1 8952.969,E2 8952.969} C_VEL
LIN {X 0,Y 617.59,Z 947.854,A -85,B 0,C 180,E1 8954.458,E2 8954.458} C_VEL
LIN {X 0,Y 620.092,Z 895.205,A -85,B 0,C 180,E1 8955.434,E2 8955.434} C_VEL
LIN {X 0,Y 619.786,Z 883.426,A -85,B 0,C 180,E1 8955.634,E2 8955.634} C_VEL
LIN {X 0,Y 595.633,Z 845.039,A -85,B 0,C 180,E1 8957.881,E2 8957.881} C_VEL
LIN {X 0,Y 577.183,Z 809.71,A -85,B 0,C 180,E1 8959.966,E2 8959.966} C_VEL
LIN {X 0,Y 577.094,Z 809.06,A -85,B 0,C 180,E1 8964.828,E2 8964.828} C_VEL
LIN {X 0,Y 577.165,Z 809.06,A -85,B 0,C 180,E1 8970.171,E2 8970.171} C_VEL
LIN {X 0,Y 577.222,Z 809.06,A -85,B 0,C 180,E1 8975.239,E2 8975.239} C_VEL
LIN {X 0,Y 577.249,Z 809.425,A -85,B 0,C 180,E1 8977.087,E2 8977.087} C_VEL
LIN {X 0,Y 596.764,Z 850.382,A -85,B 0,C 180,E1 8980.523,E2 8980.523} C_VEL
LIN {X 0,Y 609.766,Z 883,A -85,B 0,C 180,E1 8983.406,E2 8983.406} C_VEL
LIN {X 0,Y 607.212,Z 907.02,A -85,B 0,C 180,E1 8984.761,E2 8984.761} C_VEL
LIN {X 0,Y 601.082,Z 948.361,A -85,B 0,C 180,E1 8987.477,E2 8987.477} C_VEL
LIN {X 0,Y 595.228,Z 986.684,A -85,B 0,C 180,E1 8990.686,E2 8990.686} C_VEL
LIN {X 0,Y 589.652,Z 1022.898,A -85,B 0,C 180,E1 8994.485,E2 8994.485} C_VEL
LIN {X 0,Y 584.888,Z 1056.148,A -85,B 0,C 180,E1 8998.889,E2 8998.889} C_VEL
LIN {X 0,Y 581.751,Z 1082.57,A -85,B 0,C 180,E1 9003.35,E2 9003.35} C_VEL
LIN {X 0,Y 579.657,Z 1103.586,A -85,B 0,C 180,E1 9007.915,E2 9007.915} C_VEL
LIN {X 0,Y 578.668,Z 1119.123,A -85,B 0,C 180,E1 9012.44,E2 9012.44} C_VEL
LIN {X 0,Y 578.155,Z 1129.248,A -85,B 0,C 180,E1 9016.707,E2 9016.707} C_VEL
LIN {X 0,Y 577.699,Z 1135.613,A -85,B 0,C 180,E1 9021.479,E2 9021.479} C_VEL
LIN {X 0,Y 577.565,Z 1136.719,A -85,B 0,C 180,E1 9026.406,E2 9026.406} C_VEL
LIN {X 0,Y 577.993,Z 1133.605,A -85,B 0,C 180,E1 9030.389,E2 9030.389} C_VEL
LIN {X 0,Y 578.406,Z 1125.302,A -85,B 0,C 180,E1 9035.079,E2 9035.079} C_VEL
LIN {X 0,Y 579.124,Z 1112.015,A -85,B 0,C 180,E1 9039.713,E2 9039.713} C_VEL
LIN {X 0,Y 580.499,Z 1093.918,A -85,B 0,C 180,E1 9044.253,E2 9044.253} C_VEL
LIN {X 0,Y 583.196,Z 1069.397,A -85,B 0,C 180,E1 9048.916,E2 9048.916} C_VEL
LIN {X 0,Y 587.009,Z 1040.642,A -85,B 0,C 180,E1 9053.206,E2 9053.206} C_VEL
LIN {X 0,Y 592.072,Z 1006.443,A -85,B 0,C 180,E1 9057.263,E2 9057.263} C_VEL
LIN {X 0,Y 597.942,Z 969.359,A -85,B 0,C 180,E1 9060.762,E2 9060.762} C_VEL
LIN {X 0,Y 604.136,Z 928.493,A -85,B 0,C 180,E1 9063.82,E2 9063.82} C_VEL
LIN {X 0,Y 609.909,Z 886.623,A -85,B 0,C 180,E1 9066.263,E2 9066.263} C_VEL
LIN {X 0,Y 609.303,Z 881.552,A -85,B 0,C 180,E1 9066.629,E2 9066.629} C_VEL
LIN {X 0,Y 594.585,Z 844.998,A -85,B 0,C 180,E1 9069.941,E2 9069.941} C_VEL
LIN {X 0,Y 577.404,Z 810.131,A -85,B 0,C 180,E1 9073.189,E2 9073.189} C_VEL
LIN {X 0,Y 577.307,Z 809.06,A -85,B 0,C 180,E1 9073.273,E2 9073.273} C_VEL
LIN {X 0,Y 577.651,Z 809.06,A -85,B 0,C 180,E1 9077.927,E2 9077.927} C_VEL
LIN {X 0,Y 577.885,Z 809.06,A -85,B 0,C 180,E1 9083.499,E2 9083.499} C_VEL
LIN {X 0,Y 577.961,Z 809.06,A -85,B 0,C 180,E1 9088.508,E2 9088.508} C_VEL
LIN {X 0,Y 577.895,Z 809.06,A -85,B 0,C 180,E1 9093.004,E2 9093.004} C_VEL
LIN {X 0,Y 577.866,Z 809.06,A -85,B 0,C 180,E1 9097.519,E2 9097.519} C_VEL
LIN {X 0,Y 577.712,Z 809.06,A -85,B 0,C 180,E1 9102.084,E2 9102.084} C_VEL
LIN {X 0,Y 577.638,Z 809.06,A -85,B 0,C 180,E1 9106.73,E2 9106.73} C_VEL
LIN {X 0,Y 577.477,Z 809.06,A -85,B 0,C 180,E1 9111.496,E2 9111.496} C_VEL
LIN {X 0,Y 577.305,Z 809.06,A -85,B 0,C 180,E1 9117.142,E2 9117.142} C_VEL
LIN {X 0,Y 577.247,Z 809.06,A -85,B 0,C 180,E1 9123.111,E2 9123.111} C_VEL
LIN {X 0,Y 577.134,Z 809.06,A -85,B 0,C 180,E1 9128.937,E2 9128.937} C_VEL
LIN {X 0,Y 577.177,Z 809.06,A -85,B 0,C 180,E1 9135.023,E2 9135.023} C_VEL
LIN {X 0,Y 577.099,Z 809.06,A -85,B 0,C 180,E1 9141.07,E2 9141.07} C_VEL
LIN {X 0,Y 577.176,Z 809.06,A -85,B 0,C 180,E1 9146.915,E2 9146.915} C_VEL
LIN {X 0,Y 577.372,Z 809.06,A -85,B 0,C 180,E1 9152.863,E2 9152.863} C_VEL
LIN {X 0,Y 577.51,Z 809.06,A -85,B 0,C 180,E1 9158.513,E2 9158.513} C_VEL
LIN {X 0,Y 577.615,Z 809.06,A -85,B 0,C 180,E1 9163.277,E2 9163.277} C_VEL
LIN {X 0,Y 577.76,Z 809.06,A -85,B 0,C 180,E1 9169.452,E2 9169.452} C_VEL
LIN {X 0,Y 577.904,Z 809.06,A -85,B 0,C 180,E1 9173.997,E2 9173.997} C_VEL
LIN {X 0,Y 578.194,Z 809.06,A -85,B 0,C 180,E1 9180.001,E2 9180.001} C_VEL
LIN {X 0,Y 577.951,Z 809.06,A -85,B 0,C 180,E1 9186.003,E2 9186.003} C_VEL
LIN {X 0,Y 577.707,Z 809.06,A -85,B 0,C 180,E1 9192.078,E2 9192.078} C_VEL
LIN {X 0,Y 577.623,Z 809.06,A -85,B 0,C 180,E1 9196.724,E2 9196.724} C_VEL
LIN {X 0,Y 577.475,Z 809.06,A -85,B 0,C 180,E1 9201.489,E2 9201.489} C_VEL
LIN {X 0,Y 577.252,Z 809.06,A -85,B 0,C 180,E1 9207.113,E2 9207.113} C_VEL
LIN {X 0,Y 577.247,Z 809.06,A -85,B 0,C 180,E1 9213.095,E2 9213.095} C_VEL
LIN {X 0,Y 577.179,Z 809.092,A -85,B 0,C 180,E1 9218.69,E2 9218.69} C_VEL
LIN {X 0,Y 579.369,Z 814.54,A -85,B 0,C 180,E1 9219.035,E2 9219.035} C_VEL
LIN {X 0,Y 603.785,Z 854.667,A -85,B 0,C 180,E1 9222.205,E2 9222.205} C_VEL
LIN {X 0,Y 621.581,Z 884.777,A -85,B 0,C 180,E1 9224.247,E2 9224.247} C_VEL
LIN {X 0,Y 619.484,Z 935.571,A -85,B 0,C 180,E1 9225.146,E2 9225.146} C_VEL
LIN {X 0,Y 615.545,Z 982.369,A -85,B 0,C 180,E1 9226.442,E2 9226.442} C_VEL
LIN {X 0,Y 614.609,Z 992.848,A -85,B 0,C 180,E1 9226.806,E2 9226.806} C_VEL
LIN {X 0,Y 609.652,Z 1009.677,A -85,B 0,C 180,E1 9227.221,E2 9227.221} C_VEL
LIN {X 0,Y 604.919,Z 1025.197,A -85,B 0,C 180,E1 9227.692,E2 9227.692} C_VEL
LIN {X 0,Y 599.739,Z 1066.079,A -85,B 0,C 180,E1 9229.848,E2 9229.848} C_VEL
LIN {X 0,Y 592.883,Z 1109.206,A -85,B 0,C 180,E1 9232.89,E2 9232.89} C_VEL
LIN {X 0,Y 586.575,Z 1147.807,A -85,B 0,C 180,E1 9236.361,E2 9236.361} C_VEL
LIN {X 0,Y 580.597,Z 1185.163,A -85,B 0,C 180,E1 9240.64,E2 9240.64} C_VEL
LIN {X 0,Y 576.288,Z 1214.283,A -85,B 0,C 180,E1 9244.857,E2 9244.857} C_VEL
LIN {X 0,Y 573.126,Z 1240.724,A -85,B 0,C 180,E1 9249.739,E2 9249.739} C_VEL
LIN {X 0,Y 571.402,Z 1259.344,A -85,B 0,C 180,E1 9254.266,E2 9254.266} C_VEL
LIN {X 0,Y 570.601,Z 1273.208,A -85,B 0,C 180,E1 9258.884,E2 9258.884} C_VEL
LIN {X 0,Y 570.334,Z 1281.69,A -85,B 0,C 180,E1 9263.108,E2 9263.108} C_VEL
LIN {X 0,Y 570.245,Z 1285.871,A -85,B 0,C 180,E1 9266.956,E2 9266.956} C_VEL
LIN {X 0,Y 570.384,Z 1286.668,A -85,B 0,C 180,E1 9271.512,E2 9271.512} C_VEL
